*********************************************************************************************************)
FUNCTION_BLOCK FB_ASI_Projecting
VAR_INPUT
	iSlaveaddress		:BYTE;
	iParametervalue		:DWORD;
	bIOValue			:BOOL;	(*Read/Write IO-value of a slave*)
	bIDCode				:BOOL;	(*Read/Write	ID-code of a slave*)
	bReadWrite			:BOOL;	(*0: Read, 1: Write*)
	bReadLPS			:BOOL;	(*Read List of all projected Slaves*)
	bStart				:BOOL;
END_VAR
VAR_OUTPUT
	bBusy				:BOOL;
	bErr					:BOOL;
	iErrornumber			:DWORD;
	iParameterReadvalue	:BYTE;	(*IO-value or ID-code of a slave*)
	iLPS				:DWORD;
END_VAR
VAR_IN_OUT
	stParameterBuffer		:ST_ParameterBuffer;
END_VAR
VAR
	iProjectingStep	:INT;
	TrigStart			:R_TRIG;
	iAddressFactor	:BYTE;
	iParameternumber	:WORD;
	iReadValue		:DWORD;
	fbParameterinterface	:FB_ASI_Parameterinterface;
END_VAR
	CASE iProjectingStep OF

	(*Idle*)
	0:	TrigStart(clk:=bStart);
		IF TrigStart.Q THEN
			bBusy				:=TRUE;
			bErr					:=FALSE;
			iErrornumber			:=0;
			iProjectingStep		:=1;
		END_IF

	(*generate Parameternumber*)
	1:	iAddressFactor	:=iSlaveaddress / 8;
		IF bIOValue THEN
			iParameternumber	:=16#40+iAddressFactor;
		ELSIF bIDCode THEN
			iParameternumber	:=16#48+iAddressFactor;
		ELSIF bReadLPS	THEN
			iParameternumber	:=16#A8;
		END_IF
		iProjectingStep	:=2;

	(*write Parameter to ASI-Master*)
	2:	fbParameterinterface(iParameternumber	:=iParameternumber,
							iParametervalue	:=iParametervalue,
							stParameterBuffer	:=stParameterBuffer,
							bParametermode	:=bReadWrite,
							bCycleMode		:=TRUE,
							bStart			:=TRUE);
			IF (NOT fbParameterinterface.bBusy)  THEN
				IF fbParameterinterface.bErr THEN
					bErr			:=TRUE;
					iErrornumber	:=fbParameterinterface.iErrornumber;
					iProjectingStep	:=10;
				ELSE
					iReadValue	:=fbParameterinterface.iParameterReadvalue;
					iProjectingStep	:=3;
				END_IF
				fbParameterinterface(bStart			:=FALSE,
								stParameterBuffer	:=stParameterBuffer);
			END_IF

	(*generate ParameterReadvalue*)
	3:	IF bReadLPS THEN
			iParameterReadvalue	:=0;
			iLPS				:=iReadValue;
		ELSE
			iParameterReadvalue	:=DWORD_TO_BYTE(SHR(iReadValue,((iSlaveaddress-iAddressFactor*8)*4))) AND 2#00001111;
			iLPS	:=0;
		END_IF
		iProjectingStep	:=10;

	(*Quit*)
	10:	bBusy			:=FALSE;
		bStart			:=FALSE;
		iProjectingStep	:=0;

	ELSE
		;
	END_CASE
END_FUNCTION_BLOCK

(* POU FB_ASI_ReadParameter, ST *)
(*********************************************************************************************************

NAME..............	:	FB_ReadParameter
DATE...............	:	21.03.2002
AUTHOR........	:	G.Sieder (Beckhoff Industrieelektronik)

DESCRIPTION:	FB to read Parameters 

HISTORY:	
21.03.2002	gs	start coding

*********************************************************************************************************)
FUNCTION_BLOCK FB_ASI_ReadParameter
VAR_INPUT
	iParameternumber		:WORD;
	bCycleMode			:BOOL;		(*0: Acyclic , 1:Cyclic (permanent Read/Write) *)
	bStart				:BOOL;
END_VAR
VAR_OUTPUT
	bBusy				:BOOL;
	bErr					:BOOL;
	iErrornumber			:DWORD;
	iParameterReadvalue	:DWORD;
END_VAR
VAR_IN_OUT
	stParameterBuffer		:ST_ParameterBuffer;
END_VAR
VAR
	iReadStep	:INT;
	TrigStart		:R_TRIG;
	fbParameterinterface	:FB_ASI_Parameterinterface;
END_VAR
CASE iReadStep OF

	(*Idle*)
	0:	TrigStart(clk:=bStart);
		IF TrigStart.Q THEN
			bBusy				:=TRUE;
			bErr					:=FALSE;
			iErrornumber			:=0;
			iReadStep			:=1;
		END_IF

	(*wite Parameters to ASI-Master*)
	1:	fbParameterinterface(iParameternumber	:=iParameternumber,
							stParameterBuffer	:=stParameterBuffer,
							bParametermode	:=FALSE,
							bCycleMode		:=bCycleMode,
							bStart			:=TRUE);
		(*read Parameters *)
		IF (NOT fbParameterinterface.bBusy) OR  bCycleMode THEN
			IF fbParameterinterface.bErr THEN
				bErr			:=TRUE;
				iErrornumber	:=fbParameterinterface.iErrornumber;
				iReadStep	:=5;
			ELSE
				iParameterReadvalue	:=fbParameterinterface.iParameterReadvalue;
				IF (NOT bCycleMode) OR (NOT bStart) THEN
					iReadStep	:=5;
				ELSE
					iReadStep	:=1;
				END_IF
			END_IF
		END_IF

	5:	fbParameterinterface(bStart			:=FALSE,
						stParameterBuffer	:=stParameterBuffer);
		IF (NOT fbParameterinterface.bBusy) THEN
			iReadStep	:=10;
		END_IF

	(*Quit*)
	10:	bBusy			:=FALSE;
		bStart			:=FALSE;
		iReadStep	:=0;

	ELSE
		;
	END_CASE
END_FUNCTION_BLOCK

(* POU FB_ASI_SlaveDiag, ST *)
(*********************************************************************************************************

NAME..............	:	FB_WriteParameter
DATE...............	:	21.03.2002
AUTHOR........	:	G.Sieder (Beckhoff Industrieelektronik)

DESCRIPTION:	FB for cyclic slave-diagnosis

HISTORY:	
21.03.2002	gs	start coding
03.09.2002	gs	replace bStop by bCycleMode
*********************************************************************************************************)
FUNCTION_BLOCK FB_ASI_SlaveDiag
VAR_INPUT
	iSlaveaddress		:BYTE;
	iCounter				:INT;		(*1:PhysicalFaultCounter,  2:TimeoutCounter,  3:ResponseCounter,  4:Leave-DataExchCounter,  5:DataExch-FailedCounter *)
	bCounterReset		:BOOL;
	bReadLES			:BOOL;		(*Read List of all detected Slaves*)
	bReadLAS			:BOOL;		(*Read List of all activated Slaves*)
	bCycleMode			:BOOL;		(*0: Acyclic , 1:Cyclic (permanent Read/Write) *)
	bStart				:BOOL;

END_VAR
VAR_OUTPUT
	bBusy				:BOOL;
	bErr					:BOOL;
	iErrornumber			:DWORD;
	iCounterValue		:WORD;		(*Counter of a slave*)
	iSlaveList			:DWORD;	(*LES or LAS of all Slaves*)
END_VAR
VAR_IN_OUT
	stParameterBuffer		:ST_ParameterBuffer;
END_VAR
VAR
	iDiagStep			:INT;
	TrigStart				:R_TRIG;
	iAddressFactor		:BYTE;
	iParameternumber		:WORD;
	iReadValue			:DWORD;
	fbParameterinterface	:FB_ASI_Parameterinterface;

	TimerResetCounter	:TON;
END_VAR
	CASE iDiagStep OF

	(*Idle*)
	0:	TrigStart(clk:=bStart);
		IF TrigStart.Q THEN
			bBusy				:=TRUE;
			bErr					:=FALSE;
			iErrornumber			:=0;
			iDiagStep			:=1;
		END_IF

	(*generate Parameternumber*)
	1:	iAddressFactor	:=iSlaveaddress / 2;
		IF bReadLES	THEN
			iParameternumber	:=16#B0;
		ELSIF bReadLAS THEN
			iParameternumber	:=16#B8;
		ELSE
			CASE iCounter OF
				1:	iParameternumber	:=16#140+iAddressFactor;
				2:	iParameternumber	:=16#160+iAddressFactor;
				3:	iParameternumber	:=16#180+iAddressFactor;
				4:	iParameternumber	:=16#1A0+iAddressFactor;
				5:	iParameternumber	:=16#1C0+iAddressFactor;
			ELSE
				;
			END_CASE
		END_IF
		iDiagStep	:=2;

	(*write Parameter to ASI-Master*)
	2:	fbParameterinterface(iParameternumber		:=iParameternumber,
							stParameterBuffer		:=stParameterBuffer,
							iParametervalue		:=0,
							bParametermode		:=bCounterReset,
							bCycleMode			:=TRUE,
							bStart				:=TRUE);
				IF fbParameterinterface.bErr THEN
					bErr			:=TRUE;
					iErrornumber	:=fbParameterinterface.iErrornumber;
					iDiagStep	:=10;
				ELSE
					iReadValue	:=fbParameterinterface.iParameterReadvalue;
					iDiagStep	:=3;
				END_IF
				TimerResetCounter(in:=bCounterReset,pt:=t#200ms);
				IF TimerResetCounter.Q THEN
					bCounterReset		:=FALSE;
					TimerResetCounter.IN 	:=FALSE;
				END_IF

	(*generate ParameterReadvalue*)
	3:	fbParameterinterface(stParameterBuffer	:=stParameterBuffer);
		IF bReadLES OR bReadLAS THEN
			iCounterValue	:=0;
			iSlaveList		:=iReadValue;
		ELSE
			iCounterValue	:=DWORD_TO_WORD(SHR(iReadValue,((iSlaveaddress-iAddressFactor*2)*16)));
			iSlaveList	:=0;
		END_IF
		IF (NOT bStart) THEN
			fbParameterinterface(bStart	:=FALSE,
							stParameterBuffer	:=stParameterBuffer);
			IF (NOT fbParameterinterface.bBusy) THEN
				iDiagStep	:=10;
			END_IF
		ELSE
			iDiagStep	:=2;
		END_IF

	(*Quit*)
	10:	bBusy		:=FALSE;
		bStart		:=FALSE;
		iDiagStep	:=0;

	ELSE
		;
	END_CASE
END_FUNCTION_BLOCK

(* POU FB_ASI_WriteParameter, ST *)
(*********************************************************************************************************

NAME..............	:	FB_WriteParameter
DATE...............	:	21.03.2002
AUTHOR........	:	G.Sieder (Beckhoff Industrieelektronik)

DESCRIPTION:	FB to write Parameters 

HISTORY:	
21.03.2002	gs	start coding
03.09.2002	gs	Output ReadValue removed
*********************************************************************************************************)
FUNCTION_BLOCK FB_ASI_WriteParameter
VAR_INPUT
	iParameternumber		:WORD;
	iParametervalue		:DWORD;
	bStart				:BOOL;
END_VAR
VAR_OUTPUT
	bBusy				:BOOL;
	bErr					:BOOL;
	iErrornumber			:DWORD;
END_VAR
VAR_IN_OUT
	stParameterBuffer		:ST_ParameterBuffer;
END_VAR
VAR
	iWriteStep	:INT;
	TrigStart		:R_TRIG;
	fbParameterinterface	:FB_ASI_Parameterinterface;
END_VAR
	CASE iWriteStep OF

	(*Idle*)
	0:	TrigStart(clk:=bStart);
		IF TrigStart.Q THEN
			bBusy				:=TRUE;
			bErr					:=FALSE;
			iErrornumber			:=0;
			iWriteStep			:=1;
		END_IF

	(*wite Parameters to ASI-Master*)
	1:	fbParameterinterface(iParameternumber	:=iParameternumber,
							iParametervalue	:=iParametervalue,
							stParameterBuffer	:=stParameterBuffer,
							bParametermode	:=TRUE,
							bCycleMode		:= FALSE,
							bStart			:=TRUE);
		IF  fbParameterinterface.bBusy  THEN
			iWriteStep	:=5;
		END_IF


	5:	fbParameterinterface(stParameterBuffer	:=stParameterBuffer);
		IF (NOT fbParameterinterface.bBusy) THEN
			IF fbParameterinterface.bErr THEN
				bErr			:=TRUE;
				iErrornumber	:=fbParameterinterface.iErrornumber;
			END_IF
			iWriteStep	:=10;
		END_IF

	(*Quit*)
	10:	bBusy			:=FALSE;
		bStart			:=FALSE;
		iWriteStep	:=0;

	ELSE
		;
	END_CASE
END_FUNCTION_BLOCK

(* POU FB_ASI_WriteReadParameter, ST *)
(*********************************************************************************************************

NAME..............	:	FB_WriteReadParameter
DATE...............	:	18.08.2003
AUTHOR........	:	G.Sieder (Beckhoff Industrieelektronik)

DESCRIPTION:	FB to write Parameters with answer 

HISTORY:	
18.08.2003	gs	start coding

*********************************************************************************************************)
FUNCTION_BLOCK FB_ASI_WriteReadParameter
VAR_INPUT
	iParameternumber		:WORD;
	iParametervalue		:DWORD;
	bStart				:BOOL;
END_VAR
VAR_OUTPUT
	bBusy				:BOOL;
	bErr					:BOOL;
	iParameterReadValue	:DWORD;
	iErrornumber			:DWORD;
END_VAR
VAR_IN_OUT
	stParameterBuffer		:ST_ParameterBuffer;
END_VAR
VAR
	iWriteStep	:INT;
	TrigStart		:R_TRIG;
	fbParameterinterface	:FB_ASI_Parameterinterface;
END_VAR
	CASE iWriteStep OF

	(*Idle*)
	0:	TrigStart(clk:=bStart);
		IF TrigStart.Q THEN
			bBusy				:=TRUE;
			bErr					:=FALSE;
			iErrornumber			:=0;
			iWriteStep			:=1;
		END_IF

	(*wite Parameters to ASI-Master*)
	1:	fbParameterinterface(iParameternumber	:=iParameternumber,
							iParametervalue	:=iParametervalue,
							stParameterBuffer	:=stParameterBuffer,
							bParametermode	:=TRUE,
							bCycleMode		:= FALSE,
							bStart			:=TRUE);
		IF  fbParameterinterface.bBusy  THEN
			iWriteStep	:=5;
		END_IF


	5:	fbParameterinterface(stParameterBuffer	:=stParameterBuffer);
		IF (NOT fbParameterinterface.bBusy) THEN
			IF fbParameterinterface.bErr THEN
				bErr			:=TRUE;
				iErrornumber	:=fbParameterinterface.iErrornumber;
				iParameterReadValue	:=0;
			ELSE
				iParameterReadValue	:=fbParameterinterface.iParameterReadvalue;
			END_IF
			iWriteStep	:=10;
		END_IF

	(*Quit*)
	10:	bBusy			:=FALSE;
		bStart			:=FALSE;
		iWriteStep	:=0;

	ELSE
		;
	END_CASE
END_FUNCTION_BLOCK

(* POU FB_AX2000_AXACT, ST *)
FUNCTION_BLOCK FB_AX2000_AXACT
VAR_INPUT
	bMode_DigitalSpeed	: BOOL;			(*OP-Mode digital speed instead of Positioning*)
	iDigitalSpeed			: DWORD;			(*digital speed if OP-Mode = digital speed*)
	iVelocity				: DWORD;		(*Velocity*)
	iPosition				: DINT;			(*Position*)
	imotion_tasknumber	: WORD;			(*number of EEPROM-saved motion-task*)
	imotion_blocktype		: WORD;			(*optional Parameters of motion tasks*)
	bStart				: BOOL;			(*START*)
	bStop				: BOOL;			(*STOP*)
	bShortStop			: BOOL;			(*1: break of motion task, 0: continue same motion task*)
	bErrorResume		: BOOL;			(*Error resume*)
	tTimeOut				: TIME:=t#5s;
END_VAR
VAR_OUTPUT

	bBusy				: BOOL;
	bError				: BOOL;			(*Errorstatus of Servo*)
	bTimeOutErr			: BOOL;

END_VAR
VAR
	i16State:				INT;
	icheckStatus:			WORD;
	icheckControlWord:	WORD;			(*ControlWord for Servo*)

	bServoReady:		BOOL;			(*readyFlag for HSW*)
	TrigStart:				R_TRIG;
	TrigTimeOut:			R_TRIG;
	bResetServo:			BOOL;			(*first move of Servo after Start/Restart*)

	TimerTimeOut		:TON;
	bTimeOutStart		:BOOL;

	iHighByte			:BYTE;
	iLowByte				:BYTE;
	icheckByteSwaping	:WORD;
	bMapInOutputs		:BOOL;
	bShortStop_check		:BOOL;

	(*virtual Input/Output*)
	stPZD_IN:		ST_PZD_IN;
	stPZD_OUT:		ST_PZD_OUT;
END_VAR
VAR_IN_OUT
	stPZDIN:		ST_PZD_IN;			(*Data from NC*)
	stPZDOUT:		ST_PZD_OUT;			(*Data to NC*)
END_VAR
	a_MapInputs();			(*mapping of real Inputs to virtual Inputs by swaping LowByte and HighByte*)
	a_RW_CtrlWord();			(*AXACT-controls*)
	a_MapOutputs();			(*mapping of virtual Outputs to real Outputs by swaping LowByte and HighByte*)
END_FUNCTION_BLOCK
ACTION a_MapInputs:
stPZD_IN.wSTW		:=ROL(stPZDIN.wSTW,8);
stPZD_IN.wHIW		:=ROL(stPZDIN.wHIW,8);
stPZD_IN.PZD3		:=ROL(stPZDIN.PZD3,8);
stPZD_IN.PZD4		:=ROL(stPZDIN.PZD4,8);
stPZD_IN.PZD5		:=ROL(stPZDIN.PZD5,8);
stPZD_IN.PZD6		:=ROL(stPZDIN.PZD6,8);
END_ACTION
ACTION a_MapOutputs:
IF bMapInOutputs THEN
	stPZDOUT.wCtrlW		:=ROL(stPZD_OUT.wCtrlW,8);
	stPZDOUT.PZD2		:=ROL(stPZD_OUT.PZD2,8);
	stPZDOUT.PZD3		:=ROL(stPZD_OUT.PZD3,8);
	stPZDOUT.PZD4		:=ROL(stPZD_OUT.PZD4,8);
	stPZDOUT.PZD5		:=ROL(stPZD_OUT.PZD5,8);
	stPZDOUT.PZD6		:=ROL(stPZD_OUT.PZD6,8);
END_IF
END_ACTION
ACTION a_RW_CtrlWord:
	bMapInOutputs	:= TRUE;

	(* Errorstatus*)
	icheckStatus:=2#00000000_00001000;
	IF (stPZD_IN.wSTW AND icheckStatus)<>0 THEN
		i16State:=10;
	END_IF

	(*short break of a motion task*)
	IF bShortStop AND (NOT bShortStop_check)THEN
		stPZD_OUT.wCtrlW:=stPZD_OUT.wCtrlW AND 2#1111111111011111;
		bShortStop_check	:=TRUE;
	ELSIF (NOT bShortStop) AND bShortStop_check THEN
		bShortStop_check	:=FALSE;
		IF (NOT bStart) THEN
			i16State			:= 11;
			bBusy			:= FALSE;
		ELSE
			stPZD_OUT.wCtrlW:=stPZD_OUT.wCtrlW OR 2#0000000000100000;
		END_IF
	END_IF

	(*Stophandling*)
	IF  bStop THEN
		stPZD_OUT.wCtrlW:=2#0000000000000101;
		bBusy			:= FALSE;
		bStart			:= FALSE;
		bMapInOutputs	:= TRUE;
		i16State			:= 11;
	END_IF

	(*TimeOut*)
	IF (NOT bMode_DigitalSpeed) THEN
		TrigTimeOut(clk:=bStart);
		IF TrigTimeOut.Q THEN
			bTimeOutStart	:=TRUE;
			bTimeOutErr		:= FALSE;
			bError			:= FALSE;
		END_IF
		IF bBusy THEN
			TimerTimeOut(IN:= FALSE, PT:= tTimeOut );
			bTimeOutStart	:=FALSE;
		ELSE
			TimerTimeOut(IN:= bTimeOutStart, PT:= tTimeOut );
		END_IF
		IF TimerTimeOut.Q THEN
			bTimeOutErr		:=TRUE;
			bTimeOutStart	:= FALSE;
			bServoReady	:= FALSE;
			i16State			:= 11;
		END_IF
	END_IF

	CASE i16State OF

		(*Initialisierung*)
	0:	bServoReady:= 	FALSE;
		bResetServo:=	TRUE;
		i16State:= i16State+1;

		(*Einschaltsperre*)
	1:	stPZD_OUT.wCtrlW:=2#0000000000000000;
		icheckStatus:=2#0000000001000000;
		IF (stPZD_IN.wSTW AND icheckStatus)<>0 THEN
			stPZD_OUT.wCtrlW:=2#0000000000000110;
			bServoReady:= FALSE;
			i16State:= i16State+1;
		END_IF

		(*einschaltbereit*)
	2:	icheckStatus:=2#0000001000000001;
		IF (stPZD_IN.wSTW AND icheckStatus)<>0 THEN
			stPZD_OUT.wCtrlW:=2#0000000000000111;
			bServoReady:= FALSE;
			i16State:= i16State+1;
		END_IF

		(*betriebsbereit*)
	3:	icheckStatus:=2#0000001000100011;
		IF (stPZD_IN.wSTW AND icheckStatus)<>0 THEN
			stPZD_OUT.wCtrlW:=2#0000010000111111;
			i16State:= i16State+1;
		END_IF

		(*Betrieb freigegeben*)
	4:	icheckStatus:=2#0000001000100111;
		IF (stPZD_IN.wSTW AND icheckStatus)<>0 THEN
			i16State:= i16State+1;
		END_IF

		(*benutzerdefinierte Daten übertragen*)
	5:	TrigStart(clk:=bStart);
		bMapInOutputs	:= FALSE;
		IF TrigStart.Q THEN
			bMapInOutputs:= TRUE;
			a_RW_PZD();
			bError		:= FALSE;
			bTimeOutErr	:= FALSE;
			bResetServo	:= FALSE;
		END_IF
		IF (NOT bResetServo) THEN
			icheckStatus:=2#0010000000000000;
			IF (stPZD_IN.wSTW AND icheckStatus)<>0 THEN
				;
			ELSE
				bBusy	:= TRUE;
				i16State:= 6;
			END_IF
		END_IF

	6:	icheckStatus:=2#0010000000000000;
		IF (stPZD_IN.wSTW AND icheckStatus)<>0 THEN
			bBusy	:= FALSE;
			i16State:= 5;
		END_IF
		IF bMode_DigitalSpeed THEN
			stPZD_OUT.PZD3	:=DWORD_TO_WORD(iDigitalSpeed*140);
			stPZD_OUT.PZD2	:=DWORD_TO_WORD(SHR((iDigitalSpeed*140),16));
		END_IF

		(* Errorhandling*)
	10:	bError			:= TRUE;
		bBusy			:= FALSE;
		bServoReady	:= FALSE;
		IF BErrorResume THEN
			stPZD_OUT.wCtrlW:=2#0000010010001111;
			i16State:=11;
		END_IF

	11:	IF (NOT bStart) THEN
			i16State:=0;
		END_IF

END_CASE
END_ACTION
ACTION a_RW_PZD:
IF bMode_DigitalSpeed THEN
	stPZD_OUT.PZD3	:=DWORD_TO_WORD(iDigitalSpeed*140);
	stPZD_OUT.PZD2	:=DWORD_TO_WORD(SHR((iDigitalSpeed*140),16));
	icheckControlWord:=2#0000000001000000;
	IF (icheckControlWord AND stPZD_OUT.wCtrlW)<>0 THEN
		stPZD_OUT.wCtrlW:=16#443F;
	ELSE
		stPZD_OUT.wCtrlW:=16#447F;
	END_IF
ELSIF (imotion_tasknumber <> 0) THEN
	stPZD_OUT.PZD2	:=imotion_tasknumber;
	icheckControlWord:=2#0000000001000000;
	IF (icheckControlWord AND stPZD_OUT.wCtrlW)<>0 THEN
		stPZD_OUT.wCtrlW:=16#043F;
	ELSE
		stPZD_OUT.wCtrlW:=16#047F;
	END_IF
ELSIF (iVelocity<>0) THEN
	stPZD_OUT.PZD3	:=DWORD_TO_WORD(iVelocity);
	stPZD_OUT.PZD2	:=DWORD_TO_WORD(SHR(iVelocity,16));
	stPZD_OUT.PZD5	:=DWORD_TO_WORD(DINT_TO_DWORD( iPosition ));
	stPZD_OUT.PZD4	:=DWORD_TO_WORD(SHR(DINT_TO_DWORD( iPosition ),16));
	stPZD_OUT.PZD6	:=imotion_blocktype;
	icheckControlWord:=2#0000000001000000;
	IF (icheckControlWord AND stPZD_OUT.wCtrlW)<>0 THEN
		stPZD_OUT.wCtrlW:=16#443F;
	ELSE
		stPZD_OUT.wCtrlW:=16#447F;
	END_IF
END_IF
END_ACTION

(* POU FB_AX2000_JogMode, ST *)
FUNCTION_BLOCK FB_AX2000_JogMode
VAR_INPUT
	bStart		: BOOL;
	bStop		: BOOL;
	iBasicVelo	: INT;				(*BasicVelocity*)
	tTimeOut		: TIME:=t#5s;

END_VAR
VAR_OUTPUT
	bBusy		: BOOL;
	bErr			: BOOL;
	bTimeOutErr	: BOOL;

END_VAR
VAR_IN_OUT
	stPZDIN			: ST_PZD_IN;			(*Data from NC*)
	stPZDOUT		: ST_PZD_OUT;		(*Data to NC*)
END_VAR
VAR
	i16state			: INT;

	icheckStatus		: DWORD;
	TrigTimeOut		: R_TRIG;
	bTimeOutStart	: BOOL;
	TimerTimeOut	: TON;
	bMapInOutputs	: BOOL;
	(*virtual Input/Output*)
	stPZD_IN:		ST_PZD_IN;
	stPZD_OUT:		ST_PZD_OUT;

END_VAR
	a_MapInputs();

	(* Errorstatus*)
	icheckStatus:=2#00000000_00001000;
	IF (stPZD_IN.wSTW AND icheckStatus)<>0 THEN
		bErr	:= TRUE;
		i16State:=10;
	END_IF

	(*TimeOut*)
	TrigTimeOut(clk:=bStart);
	IF TrigTimeOut.Q THEN
		bTimeOutStart	:=TRUE;
	END_IF
	IF bBusy THEN
		TimerTimeOut(IN:= FALSE, PT:= tTimeOut );
		bTimeOutStart	:=FALSE;
	ELSE
		TimerTimeOut(IN:= bTimeOutStart, PT:= tTimeOut );
	END_IF
	IF TimerTimeOut.Q THEN
		TimerTimeOut(IN:= FALSE, PT:= tTimeOut );
		bTimeOutErr		:=TRUE;
		bTimeOutStart	:= FALSE;
		i16State			:= 10;
	END_IF

	CASE i16state OF

	0:	IF bStart THEN
			bErr				:= FALSE;
			bTimeOutErr		:= FALSE;
			i16state			:= 1;
		END_IF

	1:	stPZD_OUT.PZD2	:=iBasicVelo;
		stPZD_OUT.wCtrlW:=(ROL(stPZDOUT.wCtrlW,8))+16#100;
		bMapInOutputs	:= TRUE;
		i16state	:= 2;

	2:	icheckStatus:=2#00100010_00000000;
		IF (stPZD_IN.wSTW AND icheckStatus)=0 OR  (stPZD_IN.wSTW AND icheckStatus)=16#2200 THEN
			;
		ELSE
			bBusy	:=TRUE;
			i16state	:= 3;
		END_IF

	3:	IF bStop THEN
			stPZD_OUT.wCtrlW:=(ROL(stPZDOUT.wCtrlW,8))-16#100;
			i16state	:= 10;
		END_IF

	10:	bBusy			:=FALSE;
		bMapInOutputs	:=FALSE;
		IF (NOT bstart) THEN
			i16state	:= 0;
		END_IF

	END_CASE

	a_MapOutputs();
END_FUNCTION_BLOCK
ACTION a_MapInputs:
	stPZD_IN.wSTW		:=ROL(stPZDIN.wSTW,8);
	stPZD_IN.wHIW		:=ROL(stPZDIN.wHIW,8);
	stPZD_IN.PZD3		:=ROL(stPZDIN.PZD3,8);
	stPZD_IN.PZD4		:=ROL(stPZDIN.PZD4,8);
	stPZD_IN.PZD5		:=ROL(stPZDIN.PZD5,8);
	stPZD_IN.PZD6		:=ROL(stPZDIN.PZD6,8);
END_ACTION
ACTION a_MapOutputs:
IF bMapInOutputs THEN
	stPZDOUT.wCtrlW		:=ROL(stPZD_OUT.wCtrlW,8);
	stPZDOUT.PZD2		:=ROL(stPZD_OUT.PZD2,8);
	stPZDOUT.PZD3		:=ROL(stPZD_OUT.PZD3,8);
	stPZDOUT.PZD4		:=ROL(stPZD_OUT.PZD4,8);
	stPZDOUT.PZD5		:=ROL(stPZD_OUT.PZD5,8);
	stPZDOUT.PZD6		:=ROL(stPZD_OUT.PZD6,8);
END_IF
END_ACTION

(* POU FB_AX2000_Parameter, ST *)
FUNCTION_BLOCK FB_AX2000_Parameter
VAR_INPUT
	iSlaveAddress:	BYTE := 0;			(* Station Address of the Slave *)
	iPnu:				WORD := 16#03A2;	(* Parameter-Number *)
	nAxis:				BYTE := 1;			(* Number of Axis *)
	iLength:			BYTE := 4;			(* Length of the parameter (2 or 4) *)
	iSubindex:			BYTE := 1;			(*Subindex*)
	iParameterValue:	DWORD := 2;			(* Parameter value *)
	iFC310xDeviceId: 	WORD := 1;			(* Device-ID of the FCxxxx *)
	bStartRead:		BOOL;				(* StartFlag to start the PKW-Read *)
	bStartWrite:		BOOL;				(* StartFlag to start the PKW-Write *)
	tTimeOut:			TIME := DEFAULT_ADS_TIMEOUT;
END_VAR
VAR_OUTPUT
	bBusy				:BOOL;
	iErrorId			:DWORD;
	iReadValue		:DINT;
END_VAR
VAR
	iError:					DWORD;
	fbReadPkw:				FB_FCxxxxDpv0PkwRead;
	fbWritePkw: 				FB_FCxxxxDpv0PkwWrite;

END_VAR
IF bStartRead OR bStartWrite THEN
	IF iLength<>2 THEN
		iLength:= 4;
	END_IF
	
	(* PKW-Read with DPV0  for Stoever-Drive (ArrayCodesNotSupported and Subindex in Octet 3 must be set) *)
	fbReadPkw(bStartFlag := bStartRead, iStationAdd := iSlaveAddress, iDeviceId := iFC310xDeviceId,nAxis := nAxis, iPnu := iPnu, iSubindex := iSubindex, iLength := iLength, bArrayCodesNotSupported := TRUE, bSubindexInOctet3 := TRUE, tTimeOut:=tTimeOut);
	IF (bStartRead AND NOT fbReadPkw.bBusy) THEN
		iError := fbReadPkw.iErrorId;
		iReadValue := fbReadPkw.iReadValue;
		bStartRead := FALSE;
	END_IF;
	
	(* PKW-Write with DPV0  for Stoever-Drive (ArrayCodesNotSupported and Subindex in Octet 3 must be set) *)
	fbWritePkw(bStartFlag := bStartWrite, iStationAdd := iSlaveAddress, iDeviceId := iFC310xDeviceId, nAxis := nAxis, iPnu := iPnu, iSubindex := iSubindex, iLength := iLength, iWriteValue := iParameterValue, bArrayCodesNotSupported := TRUE, bSubindexInOctet3 := TRUE, tTimeOut:=tTimeOut);
	IF (bStartWrite AND NOT fbWritePkw.bBusy) THEN
		iError := fbWritePkw.iErrorId;
		bStartWrite := FALSE;
	END_IF;

	bBusy:=fbReadPkw.bBusy OR fbWritePkw.bBusy;
	iErrorId:=iError;
	(*iReadValue:=iParameterValue;*)
END_IF
END_FUNCTION_BLOCK

(* POU FB_FCxxxxDpv0PkwRead, ST *)
FUNCTION_BLOCK FB_FCxxxxDpv0PkwRead
VAR_INPUT
	bStartFlag:BOOL;					(* StartFlag to start the PKW-Read *)
	iStationAdd: BYTE;				(* Station Address of the Slave *)
	iDeviceId: WORD;					(* Device-ID of the FCxxxx *)
	nAxis: BYTE;						(* Number of Axis *)
	iPnu: WORD;						(* Parameter-Number *)
	iSubindex: BYTE;					(* Subindex  *)
	iLength:BYTE;					(* Length of the parameter (2 or 4) *)
	bArrayCodesNotSupported: BOOL;	(* if the drive does not support the ARRAY-AKs 6,7 and 8, this flag should be set (then the AKs 1,2,3 will be used for Arrays) *)
	bSubindexInOctet3:BOOL;			(* if the drive needs the subindex in Octet 3 (ProfiDrive 2.0), this flag should be set *)
	tTimeOut		: TIME;
END_VAR
VAR_OUTPUT
	bBusy:BOOL;			(* Reading is busy *)
	iErrorId:DWORD;
	iReadValue:DWORD;	(* Parameter value *)
END_VAR
VAR
	fbRead:ADSREAD;
	fbDevNetId:IOF_GetDeviceNetId;
	istate:WORD := 0;
	sDevNetId:STRING(23);
	iIdxGrp: DWORD;
	iport:WORD;
	iParameterValue:DWORD;
END_VAR
CASE istate OF

	0:	(*Idle*)
		IF bStartFlag THEN
			bBusy	:=TRUE;
			istate := 1;
		END_IF

	1:	(* Get Net-ID of FCxxxx-Device *)
		fbDevNetId(NETID := '', DEVICEID := iDeviceId, START := TRUE,  TMOUT := T#1s);
		IF (NOT fbDevNetId.BUSY) THEN
			IF (NOT fbDevNetId.Err) THEN
				sDevNetId := fbDevNetId.DeviceNetId;
				istate := 2;
			ELSE
				iErrorId		:=fbDevNetId.ERRID;
				bStartFlag	:=FALSE;
				bBusy		:=FALSE;
				istate := 0;
			END_IF
			fbDevNetId(NETID := '', DEVICEID := iDeviceId, START := FALSE,  TMOUT := T#1s);
		END_IF

	2:	(* Read Parameter if StartFlag is set *)
		iport := iStationAdd;
		iport := iport + 16#1000;
		iIdxGrp := nAxis;
		iIdxGrp := SHL(iIdxGrp, 28);
		iIdxGrp := iIdxGrp +iPnu;
		IF (bArrayCodesNotSupported) THEN
			iIdxGrp := iIdxGrp + 16#8000000;
		END_IF
		IF (bSubindexInOctet3) THEN
			iIdxGrp := iIdxGrp + 16#4000000;
		END_IF
		fbRead(	NETID := sDevNetId, PORT := iport, IDXGRP := iIdxGrp, IDXOFFS := iSubindex, LEN := iLength,
				DESTADDR := ADR(iParameterValue), READ := bStartFlag, TMOUT := tTimeOut);
		istate := 3;

	3:	fbRead(	NETID := sDevNetId, PORT := iport, IDXGRP := iIdxGrp, IDXOFFS := iSubindex, LEN := iLength,
				DESTADDR := ADR(iParameterValue), READ := bStartFlag, TMOUT := tTimeOut);
		IF (NOT FbRead.BUSY) OR fbRead.Err THEN
			iErrorId := FbRead.ERRID;
			iReadValue := iParameterValue;
			istate := 4;
		END_IF

	4:	(* There must be a rising edge on the READ-input of ADSREAD to start the next reading *)
		fbRead(	NETID := sDevNetId, PORT := iport, IDXGRP := iIdxGrp, IDXOFFS := iSubindex, LEN := iLength,
				DESTADDR := ADR(iParameterValue), READ := FALSE, TMOUT := tTimeOut);
		bBusy 		:= FALSE;
		bStartFlag	:= FALSE;
		istate := 0;
END_CASE
END_FUNCTION_BLOCK

(* POU IOF_GetDeviceNetId, ST *)
FUNCTION_BLOCK IOF_GetDeviceNetId
VAR_INPUT
	NETID			: T_AmsNetId;
	DEVICEID		: UDINT;
	START			: BOOL;
	TMOUT		: TIME := DEFAULT_ADS_TIMEOUT;
END_VAR
VAR_OUTPUT
	BUSY			: BOOL;
	ERR			: BOOL;
	ERRID			: UDINT;
	DeviceNetId	: T_AmsNetId;
END_VAR
VAR
	ADSREADEX1	: ADSREADEX;
	RisingEdge	: R_TRIG;
	state			: BYTE;
	tmpNetId		: ARRAY[0..5] OF BYTE;
END_VAR
RisingEdge( CLK:=START );
IF RisingEdge.Q THEN
	state := 1;
END_IF
CASE state OF
	0:;(* idle state *)
	1:
		BUSY := TRUE;
		ERR := FALSE;
		ERRID := 0;
		DeviceNetId := '';
		MEMSET( ADR( tmpNetId ), 0, SIZEOF( tmpNetId ) );
		IF ( DEVICEID > 0 ) THEN
			ADSREADEX1( READ:=FALSE );
			ADSREADEX1( NETID:=NETID, PORT:= AMSPORT_R0_IO,
						IDXGRP:= 16#00005000 + DEVICEID, IDXOFFS:= 16#00000005,
						LEN:= SIZEOF( tmpNetId ), DESTADDR:= ADR( tmpNetId ),
						READ:=TRUE, TMOUT:= TMOUT );
			state := 2;
		ELSE
			ERR := TRUE;
			ERRID :=16#706;	(* Parameter value not correct! *)
			state := 100;
		END_IF
	2:
		ADSREADEX1( READ:=FALSE, BUSY=>BUSY, ERR=>ERR, ERRID=>ERRID );
		IF NOT BUSY THEN
			IF NOT ERR THEN
				IF ( ADSREADEX1.COUNT_R = SIZEOF( tmpNetId ) ) THEN (* check the read data length *)
					DeviceNetId := F_CreateAmsNetId( tmpNetid );
				ELSE
					ERR := TRUE;
					ERRID := 16#70B; (* 1803 invalid parameter value(s) *)
				END_IF
			END_IF
			state := 0;
		END_IF
	100:(* error state *)
		BUSY := FALSE;
		state := 0;
END_CASE
END_FUNCTION_BLOCK

(* POU FB_FCxxxxDpv0PkwWrite, ST *)
FUNCTION_BLOCK FB_FCxxxxDpv0PkwWrite
VAR_INPUT
	bStartFlag:BOOL;		(* StartFlag to start the PKW-REad *)
	iStationAdd: BYTE;		(* Station Address of the Slave *)
	iDeviceId: WORD;		(* Device-ID of the FCxxxx *)
	nAxis: BYTE;			(* Number of Axis *)
	iPnu: WORD;			(* Parameter-Number *)
	iSubindex: BYTE;		(* Subindex  *)
	iLength:BYTE;			(* Length of the parameter (2 or 4) *)
	iWriteValue:DWORD;	(* Parameter value *)
	bArrayCodesNotSupported: BOOL;	(* if the drive does not support the ARRAY-AKs 6,7 and 8, this flag should be set (then the AKs 1,2,3 will be used for Arrays) *)
	bSubindexInOctet3:BOOL;				(* if the drive needs the subindex in Octet 3 (ProfiDrive 2.0), this flag should be set *)
	tTimeOut		: TIME:=T#10s;
END_VAR
VAR_OUTPUT
	bBusy:BOOL;			(* Writing is busy *)
	iErrorId:DWORD;
END_VAR
VAR
	fbWrite:ADSWRITE;
	fbDevNetId:IOF_GetDeviceNetId;
	istate:WORD := 0;
	sDevNetId:STRING(23);
	iIdxGrp: DWORD;
	iport:WORD;
	iParameterValue:DWORD;
END_VAR
CASE istate OF

	0:	(*Idle*)
		IF bStartFlag THEN
			bBusy	:=TRUE;
			istate := 1;
		END_IF

	1:	(* Get Net-ID of FCxxxx-Device *)
		fbDevNetId(NETID := '', DEVICEID :=iDeviceId, START := TRUE,  TMOUT := T#1s);
		istate := 2;

	2:	fbDevNetId();
		IF (NOT fbDevNetId.BUSY) THEN
			IF (NOT fbDevNetId.Err) THEN
				sDevNetId := fbDevNetId.DeviceNetId;
				istate := 3;
			ELSE
				iErrorId		:=fbDevNetId.ERRID;
				bBusy		:=FALSE;
				bStartFlag	:=FALSE;
				istate := 0;
			END_IF
			fbDevNetId(NETID := '', DEVICEID := iDeviceId, START := FALSE,  TMOUT := T#1s);
		END_IF

	3:	(* Read Parameter if StartFlag is set *)
		iport := iStationAdd;
		iport := iport + 16#1000;
		iIdxGrp :=nAxis;
		iIdxGrp := SHL(iIdxGrp, 28);
		iIdxGrp := iIdxGrp + iPnu;
		IF (bArrayCodesNotSupported) THEN
			iIdxGrp := iIdxGrp + 16#8000000;
		END_IF
		IF (bSubindexInOctet3) THEN
			iIdxGrp := iIdxGrp + 16#4000000;
		END_IF
		iParameterValue :=iWriteValue;
		fbWrite(	NETID := sDevNetId, PORT := iport, IDXGRP := iIdxGrp, IDXOFFS := iSubindex, LEN := iLength,
				SRCADDR := ADR(iParameterValue), WRITE := bStartFlag, TMOUT := tTimeOut);
		istate := 4;

	4:	fbWrite();
		IF (NOT fbWrite.BUSY) OR fbWrite.Err THEN
			iErrorId := fbWrite.ERRID;
			istate := 5;
		END_IF

	5:	(* There must be a rising edge on the READ-input of ADSREAD to start the next reading *)
		fbWrite(	NETID := sDevNetId, PORT := iport, IDXGRP := iIdxGrp, IDXOFFS := iSubindex, LEN := iLength,
				SRCADDR := ADR(iParameterValue), WRITE := FALSE, TMOUT := tTimeOut);
		bBusy 		:= FALSE;
		bStartFlag	:= FALSE;
		istate := 0;
END_CASE
END_FUNCTION_BLOCK

(* POU FB_AX2000_Reference, ST *)
FUNCTION_BLOCK FB_AX2000_Reference
VAR_INPUT
	bSetRefPoint	: BOOL;		(* set Reference Point*)
	bCalibrStart	: BOOL;		(* start home running*)
	bCalibrStop	: BOOL;		(* stop home running*)
	iCalVelo		: WORD;		(* basic velocity of Calibration*)

END_VAR
VAR_OUTPUT
	bBusy	: BOOL;
	bErr	: BOOL;

END_VAR
VAR_IN_OUT
	stPZDIN		: ST_PZD_IN;	(*Data from NC*)
	stPZDOUT		: ST_PZD_OUT;(*Data to NC*)
END_VAR
VAR
	icheckStatus		: WORD;
	i16State			: INT;
	bMapInOutputs	: BOOL;
	(*virtual Input/Output*)
	stPZD_IN		: ST_PZD_IN;	(*Data from NC*)
	stPZD_OUT		: ST_PZD_OUT;(*Data to NC*)
END_VAR
	a_MapInputs();

	(* Errorstatus*)
	icheckStatus:=2#00000000_00001000;
	IF (stPZD_IN.wSTW AND icheckStatus)<>0 THEN
		i16State	:=9;
	END_IF

	CASE i16State OF

	(*start FB*)
	0:	IF bSetRefPoint OR bCalibrStart THEN
			bBusy			:= TRUE;
			bErr				:= FALSE;
			IF bSetRefPoint THEN
				i16State	:= 1;
			ELSE
				i16State	:= 3;
			END_IF
		END_IF

	(* set Reference Point *)
	1:	bMapInOutputs	:=TRUE;
		(*realization of a rising edge to set a nwe reference point*)
		stPZD_OUT.wCtrlW:=(ROL(stPZDOUT.wCtrlW,8))-16#1000;
		i16State		:= 2;

	2:	stPZD_OUT.wCtrlW:=(ROL(stPZDOUT.wCtrlW,8))+16#1000;
		i16State		:= 10;

	(* start home running*)
	3:	bMapInOutputs	:=TRUE;
		stPZD_OUT.PZD2	:=iCalVelo;
		(*stPZD_OUT.wCtrlW:=(ROL(stPZDOUT.wCtrlW,8))+16#800;*)
		stPZD_OUT.wCtrlW:=((ROL(stPZDOUT.wCtrlW,8)) OR 2#0000100000000000);
		icheckStatus:=2#0000010000000000;
		IF (stPZD_IN.wSTW AND icheckStatus)<>0 THEN
			(*Stophandling*)
			IF bCalibrStop THEN
				(*stPZD_OUT.wCtrlW:=(ROL(stPZDOUT.wCtrlW,8))-16#800;*)
				stPZD_OUT.wCtrlW:=((ROL(stPZDOUT.wCtrlW,8)) AND 2#1111011111111111);
				i16State	:= 10;
			ELSE
				;
			END_IF
		ELSE
			i16State:=4;
		END_IF

	4:	icheckStatus:=2#0000010000000000;
		IF ((stPZD_IN.wSTW AND icheckStatus)<>0)  THEN
			i16State	:= 10;
		END_IF
		(*Stophandling*)
		IF bCalibrStop THEN
			stPZD_OUT.wCtrlW:=(ROL(stPZDOUT.wCtrlW,8))-16#800;
			i16State	:= 10;
		END_IF

		(*Errorcase*)
	9:	bErr			:= TRUE;
		i16State		:= 10;

	10:	bbusy			:= FALSE;
		bMapInOutputs	:= FALSE;
		bSetRefPoint		:= FALSE;
		IF (NOT bSetRefPoint) AND (NOT bCalibrStart) THEN
			i16State	:= 0;
		END_IF

	END_CASE

	a_MapOutputs();
END_FUNCTION_BLOCK
ACTION a_MapInputs:
	stPZD_IN.wSTW		:=ROL(stPZDIN.wSTW,8);
	stPZD_IN.wHIW		:=ROL(stPZDIN.wHIW,8);
	stPZD_IN.PZD3		:=ROL(stPZDIN.PZD3,8);
	stPZD_IN.PZD4		:=ROL(stPZDIN.PZD4,8);
	stPZD_IN.PZD5		:=ROL(stPZDIN.PZD5,8);
	stPZD_IN.PZD6		:=ROL(stPZDIN.PZD6,8);
END_ACTION
ACTION a_MapOutputs:
IF bMapInOutputs THEN
	stPZDOUT.wCtrlW		:=ROL(stPZD_OUT.wCtrlW,8);
	stPZDOUT.PZD2		:=ROL(stPZD_OUT.PZD2,8);
	stPZDOUT.PZD3		:=ROL(stPZD_OUT.PZD3,8);
	stPZDOUT.PZD4		:=ROL(stPZD_OUT.PZD4,8);
	stPZDOUT.PZD5		:=ROL(stPZD_OUT.PZD5,8);
	stPZDOUT.PZD6		:=ROL(stPZD_OUT.PZD6,8);
END_IF
END_ACTION

(* POU FB_AX200X_Profibus, ST *)
FUNCTION_BLOCK FB_AX200X_Profibus
VAR_INPUT
	bInit					: BOOL;			(*Initialization*)
	bMode_DigitalSpeed	: BOOL;			(*OP-Mode digital speed instead of Positioning*)
	iDigitalSpeed			: DINT;			(*digital speed if OP-Mode = digital speed*)
	iVelocity				: DWORD;		(*Velocity*)
	iPosition				: DINT;			(*Position*)
	iRunningMode		: BYTE;			(*0:digital speed, 1: motiontask, 2: JogMode, 3: Calibration*)
	imotion_tasknumber	: WORD;			(*number of EEPROM-saved motion-task*)
	imotion_blocktype		: WORD:=16#2000;	(*optional Parameters of motion tasks, default:SI-values*)
	iJogModeBasicValue	: INT;			(*BasicVelocity for JogMode*)
	iCalVelo				: WORD;			(* basic velocity of Calibration*)
	bSetRefPoint			: BOOL;			(* set Reference Point*)
	bStart					: BOOL;			(*START*)
	bStop					: BOOL;			(*STOP*)
	bShortStop			: BOOL;			(* break of motion task*)
	iSlaveAddress			: BYTE;			(* Station Address of the Slave *)
	iFC310xDeviceId 		: WORD;			(* Device-ID of the FCxxxx *)
	bErrorResume		: BOOL;			(*Error resume*)
	tTimeOut				: TIME := DEFAULT_ADS_TIMEOUT;
END_VAR
VAR_OUTPUT

	bBusy				: BOOL;
	bError				: BOOL;			(*Errorstatus of Servo*)
	iErrID				: DWORD;
	bTimeOutErr		: BOOL;
	bInitOK			: BOOL;				(*Initialization OK*)
	iactPosition		 : DINT;		(*actual Position SI-value*)
END_VAR
VAR_IN_OUT
	stPZD_IN:			ST_PZD_IN;				(*Data from NC*)
	stPZD_OUT:			ST_PZD_OUT;			(*Data to NC*)
END_VAR
VAR
	istate					:INT;
	TimerPosition				:TON;
	fbAX2000_AXACT			: FB_AX2000_AXACT;
	fbAX2000_Parameter		: FB_AX2000_Parameter;
	fbAX2000_JogMode		: FB_AX2000_JogMode;
	fbAX2000_Reference		: FB_AX2000_Reference;

	iOPMode				:DWORD;
END_VAR
VAR CONSTANT
	(*Errors*)
	ERR_OPMODE	:DWORD:=1;

END_VAR
		fbAX2000_AXACT(bMode_DigitalSpeed	:=bMode_DigitalSpeed,
						iDigitalSpeed			:=iDigitalSpeed,
						iVelocity				:=iVelocity,
						 iPosition				:=iPosition ,
						 imotion_tasknumber	:=imotion_tasknumber ,
						 imotion_blocktype	:=imotion_blocktype ,
						bShortStop			:=bShortStop,
						 bErrorResume		:=bErrorResume ,
						 tTimeOut			:=tTimeOut ,
						stPZDIN				:= stPZD_IN,
						stPZDOUT			:=stPZD_OUT);
	IF iRunningMode<2 OR bInit THEN
			fbAX2000_AXACT.bStart	:=bStart;
	END_IF

	IF (NOT bInit) THEN
		fbAX2000_AXACT.bStop	:=bStop;
	END_IF

	IF fbAX2000_AXACT.stPZD_IN.wSTW =0 THEN
		bInitOK	:=FALSE;
	END_IF

	CASE istate OF

	(*action-mode*)
	0:	(*Initialization*)
		IF bInit THEN
			bBusy		:=TRUE;
			bError		:=FALSE;
			bTimeOutErr	:=FALSE;
			iErrID		:=0;
			bInitOK		:=FALSE;
			IF bMode_DigitalSpeed THEN
				iOPMode	:= 1;
			ELSE
				iOPMode	:= 2;
			END_IF
			istate		:=1;
		(*JogMode*)
		ELSIF iRunningMode=2 AND bStart THEN
			IF bInitOK THEN
				bBusy		:=TRUE;
				bError		:=FALSE;
				bTimeOutErr	:=FALSE;
				iErrID		:=0;
				istate		:=20;
			ELSE
				iErrID	:=ERR_OPMODE;
				istate	:=100;
			END_IF
		(*CalibrationMode*)
		ELSIF iRunningMode=3 AND (bStart OR  bSetRefPoint)THEN
			IF bInitOK THEN
				bBusy		:=TRUE;
				bError		:=FALSE;
				bTimeOutErr	:=FALSE;
				iErrID		:=0;
				istate		:=30;
			ELSE
				iErrID	:=ERR_OPMODE;
				istate	:=100;
			END_IF
		(*motion-task start*)
		ELSIF (iRunningMode=1 OR iRunningMode=0) AND bStart  THEN
			IF bInitOK THEN
				bBusy		:=TRUE;
				bError		:=FALSE;
				bTimeOutErr	:=FALSE;
				iErrID		:=0;
				istate		:=10;
			ELSE
				iErrID	:=ERR_OPMODE;
				istate	:=100;
			END_IF
		ELSIF iRunningMode>3 AND bStart  THEN
			iErrID	:=ERR_OPMODE;
			istate	:=100;
		END_IF

	(*Init*)
	1:	fbAX2000_AXACT.bStop	:=TRUE;
		istate	:=2;

	2:	fbAX2000_Parameter(iSlaveAddress:= iSlaveAddress,
						iPnu:= 930,
						iParameterValue:= iOPMode,
						iFC310xDeviceId:=iFC310xDeviceId ,
						bStartWrite:= TRUE );
		istate	:=3;

	3:	fbAX2000_Parameter();
		IF (NOT fbAX2000_Parameter.bBusy) THEN
			IF fbAX2000_Parameter.iErrorId<>0 THEN
				iErrID	:=fbAX2000_Parameter.iErrorId;
				bInit		:=FALSE;
				istate	:=100;
			ELSE
				istate	:=4;
			END_IF
			fbAX2000_AXACT.bStop	:=FALSE;
		END_IF

	4:	fbAX2000_Parameter(iSlaveAddress:= iSlaveAddress,
						iPnu:= 930,
						iFC310xDeviceId:=iFC310xDeviceId ,
						bStartRead:= TRUE );
		istate	:=5;

	5:	fbAX2000_Parameter();
		IF (NOT fbAX2000_Parameter.bBusy)  THEN
			IF fbAX2000_Parameter.iErrorId<>0 THEN
				iErrID	:=fbAX2000_Parameter.iErrorId;
				istate	:=100;
			ELSE
				bInitOK	:=TRUE;
				istate	:=110;
			END_IF
			bInit		:=FALSE;
		END_IF

	(*motion task start*)
	10:	IF fbAX2000_AXACT.bBusy THEN
			istate	:=11;
		ELSIF fbAX2000_AXACT.bError THEN
			fbAX2000_Parameter(iSlaveAddress:= iSlaveAddress,
							iPnu:= 1001,
							iFC310xDeviceId:=iFC310xDeviceId ,
							bStartRead:= TRUE );
			iErrID	:=fbAX2000_Parameter.iReadValue;
			istate	:=100;
		ELSIF fbAX2000_AXACT.bTimeOutErr  THEN
			bTimeOutErr	:=TRUE;
			istate	:=100;
		END_IF

	11:	fbAX2000_Parameter(iSlaveAddress:= iSlaveAddress,
						iPnu:= 1403,
						iFC310xDeviceId:=iFC310xDeviceId ,
						bStartRead:= TRUE);
		iactPosition	:=fbAX2000_Parameter.iReadValue;
		IF (NOT fbAX2000_AXACT.bBusy) THEN
			TimerPosition(in:=TRUE, PT:=t#1s);
			IF TimerPosition.Q THEN
				TimerPosition(in:=FALSE);
				istate	:=12;
			END_IF
		END_IF

	12:	fbAX2000_Parameter();
		iactPosition	:=fbAX2000_Parameter.iReadValue;
		IF (NOT fbAX2000_Parameter.bBusy) THEN
			istate	:=110;
		END_IF

	(*JogMode*)
	20:	fbAX2000_JogMode(bStart:= bStart,
						bStop		:= bStop,
						 iBasicVelo	:=iJogModeBasicValue,
						 tTimeOut	:=tTimeOut ,
						stPZDIN		:= stPZD_IN,
						stPZDOUT	:=stPZD_OUT);
		fbAX2000_Parameter(iSlaveAddress:= iSlaveAddress,
						iPnu:= 1403,
						iFC310xDeviceId:=iFC310xDeviceId ,
						bStartRead:= TRUE);
		iactPosition	:=fbAX2000_Parameter.iReadValue;
		IF bStop OR fbAX2000_JogMode.bErr OR fbAX2000_JogMode.bTimeOutErr THEN
			istate	:=21;
		END_IF

	21:	fbAX2000_Parameter();
		iactPosition	:=fbAX2000_Parameter.iReadValue;
		IF (NOT fbAX2000_Parameter.bBusy) THEN
			bStart		:= FALSE;
			fbAX2000_JogMode(bStart		:= bStart,
							bStop		:= FALSE,
							 iBasicVelo	:=iJogModeBasicValue,
							 tTimeOut	:=tTimeOut ,
							stPZDIN		:= stPZD_IN,
							stPZDOUT	:=stPZD_OUT);
			istate	:=110;
			IF fbAX2000_JogMode.bErr THEN
				fbAX2000_Parameter(iSlaveAddress:= iSlaveAddress,
								iPnu:= 1001,
								iFC310xDeviceId:=iFC310xDeviceId ,
								bStartRead:= TRUE );
				iErrID	:=fbAX2000_Parameter.iReadValue;
				istate	:=100;
			ELSIF fbAX2000_JogMode.bTimeOutErr THEN
				bTimeOutErr	:=TRUE;
			END_IF
		END_IF

	(*CalibrationMode*)
	30:	fbAX2000_Reference(bSetRefPoint	:= bSetRefPoint ,
						bCalibrStart		:= bStart,
						bCalibrStop		:= bStop,
						iCalVelo			:= iCalVelo,
						stPZDIN			:= stPZD_IN,
						stPZDOUT		:=stPZD_OUT);
		fbAX2000_Parameter(iSlaveAddress:= iSlaveAddress,
						iPnu:= 1403,
						iFC310xDeviceId:=iFC310xDeviceId ,
						bStartRead:= TRUE);
		iactPosition	:=fbAX2000_Parameter.iReadValue;
		IF bStop OR fbAX2000_Reference.bErr  THEN
			istate	:=31;
		END_IF

	31:	fbAX2000_Parameter();
		iactPosition	:=fbAX2000_Parameter.iReadValue;
		IF (NOT fbAX2000_Parameter.bBusy) THEN
			bStart		:= FALSE;
			fbAX2000_Reference(bCalibrStart	:= bStart,
							bCalibrStop		:= TRUE,
							stPZDIN			:= stPZD_IN,
							stPZDOUT		:=stPZD_OUT);
			istate	:=110;
			IF fbAX2000_Reference.bErr THEN
				fbAX2000_Parameter(iSlaveAddress:= iSlaveAddress,
								iPnu:= 1001,
								iFC310xDeviceId:=iFC310xDeviceId ,
								bStartRead:= TRUE );
				iErrID	:=fbAX2000_Parameter.iReadValue;
				istate	:=100;
			END_IF
		END_IF


	(*Error*)
	100:	bError	:=TRUE;
		istate	:=110;

	(*Quit*)
	110:	bBusy	:=FALSE;
		IF (NOT bStart) AND (NOT bInit) THEN
			istate	:=0;
		END_IF


	ELSE
		;
	END_CASE
END_FUNCTION_BLOCK

(* POU FB_Dpv1Read, ST *)
FUNCTION_BLOCK FB_Dpv1Read
(*****************************************************************************************************************
	DESCRIPTION:	This FUNCTION block implements DPV1 Parameter Read

	CHANGE LOG:
	BY		DATE		DESCRIPTION OF CHANGE
	ICh		2008/04/02	delay resend request after fault for 100ms
	ICh		2007/01/08	resend request after fault
	ICh		2007/01/05	iRequestRef limited to 128
	ICh		2006/08/09	wait timer decreased, bugfix for errors
	ICh		2006/07/12	Bugfix iRequestRef as VAR_IN_OUT
	ICh		2006/07/10	Bugfix for evaluate response; enhanced error reporting
	ICh		2006/07/05	First Version

******************************************************************************************************************)
VAR_INPUT
	bExecute			: BOOL;

	(* drive access info *)
	aNetId				: T_AmsNetId;	(* NetID of Profibus Master FC310x/EL6731 *)
	iProfibusSlaveAdr	: USINT;	 	(* DP address of ProfiDrive *)
	iDriveId			: USINT;		(* 0..255 possible *)
	pDpv1ReqData		: POINTER TO ARRAY [1..iMAX_DPV1_SIZE] OF BYTE;
	iDpv1ReqDataLen		: UDINT;
	pDpv1ResData		: POINTER TO ARRAY [1..iMAX_DPV1_SIZE] OF BYTE;
	iDpv1ResDataLen		: UDINT;
	tTmOut				: TIME := DEFAULT_ADS_TIMEOUT;
END_VAR
VAR_OUTPUT
	bBusy				: BOOL;
	bError				: BOOL;
	bErrorValues		: BOOL;
	iErrId				: UDINT;
	iErrorClass			: BYTE;
	iErrorCode			: BYTE;
END_VAR
VAR_IN_OUT
	iRequestRef			: USINT;		(* 1..127;    0: reserved *)
END_VAR
VAR
	fbWriteAccessData 	: ADSWRITE;
	fbReadData 			: ADSREAD;
	iState				: INT;
	bExecute_			: BOOL;

	stDpv1ReqHeader		: ST_Dpv1Header;
	stDpv1ResHeader		: ST_Dpv1Header;

	WaitTimer			: TON := (PT := T#100ms);
	TmOutTimer			: TON;
END_VAR
TmOutTimer();

CASE iState OF
0:	(* idle until rising edge on bExecute *)
	IF bExecute AND NOT bExecute_ THEN
		(* generate request reference *)
		iRequestRef := UINT_TO_USINT((USINT_TO_UINT(iRequestRef) + 1) MOD 128);
		IF iRequestRef = 0 THEN
			iRequestRef := 1;
		END_IF
		pDpv1ReqData^[1] := iRequestRef;
		MEMCPY(ADR(stDpv1ReqHeader), pDpv1ReqData, SIZEOF(stDpv1ReqHeader));

		(* clear response data *)
		MEMSET(pDpv1ResData, 0, iMAX_DPV1_SIZE);

		(* on rising edge *)
		bExecute_ 	:= bExecute;
		bBusy		:= TRUE;
		bError		:= FALSE;
		bErrorValues:= FALSE;
		iErrId		:= 0;
		iErrorClass	:= 0;
		iErrorCode	:= 0;

		(* complete read request timeout 12 times the ADS timeout *)
		TmOutTimer(IN := FALSE, PT := MAX(tTmOut * 12, T#30s));
		TmOutTimer(IN := TRUE);

		(* send request *)
		fbWriteAccessData(
			NETID	:= aNetId,
			PORT	:= 16#1000 + iProfibusSlaveAdr,
			IDXGRP	:= 0,
			IDXOFFS	:= 47,
			LEN		:= MIN(iDpv1ReqDataLen, iMAX_DPV1_SIZE),
			SRCADDR	:= pDpv1ReqData,
			WRITE	:= FALSE,
			TMOUT	:= tTmOut
		);
		fbWriteAccessData(WRITE	:= TRUE);

		iState := 1;
	END_IF

1:	(* write access data for DPV1 read request *)
	fbWriteAccessData(WRITE	:= FALSE);

	IF NOT fbWriteAccessData.BUSY THEN
		fbWriteAccessData(WRITE	:= FALSE);

		IF NOT fbWriteAccessData.ERR THEN
			(* read request parameter successfully sent, check for response *)
			WaitTimer(IN := FALSE);
			iState	:= 2; (* wait before polling *)
		ELSE
			bBusy	:= FALSE;
			bError	:= TRUE;
			iErrId	:= fbWriteAccessData.ERRID;
			IF ((UDINT_TO_DWORD(iErrId) AND DWORD#16#FF000000) = DWORD#16#27000000) THEN
				iErrorClass := UDINT_TO_BYTE(SHR((UDINT_TO_DWORD(iErrId) AND 16#00F00000), 20));
				iErrorCode := UDINT_TO_BYTE(SHR((UDINT_TO_DWORD(iErrId) AND 16#000F0000), 16));
			END_IF
			iState	:= 0;
		END_IF
	END_IF

2:	(* wait staate before next read response check *)
	WaitTimer(IN := TRUE);
	IF WaitTimer.Q THEN
		(* read request parameter successfully sent, check for read response *)
		MEMSET(pDpv1ResData, 0, iMAX_DPV1_SIZE);
		fbReadData(
			NETID	:= aNetId,
			PORT	:= 16#1000 + iProfibusSlaveAdr,
			IDXGRP	:= 0,
			IDXOFFS	:= 47,
			LEN		:= iMAX_DPV1_SIZE,
			DESTADDR:= pDpv1ResData,
			READ	:= FALSE,
			TMOUT	:= tTmOut,
		);
		fbReadData(READ := TRUE);
		iState	:= 3; (* CHECK READ *)
	END_IF

3:	(* wait for read response with data from DPV1 read request *)
	fbReadData(READ := FALSE);

	IF NOT fbReadData.BUSY THEN
		fbReadData(READ := FALSE);
		IF NOT fbReadData.ERR THEN
			MEMCPY(ADR(stDpv1ResHeader), pDpv1ResData, SIZEOF(stDpv1ResHeader));

			(* check for read response reference *)
			IF (stDpv1ResHeader.iRequestRef = stDpv1ReqHeader.iRequestRef) AND (stDpv1ResHeader.iAxis = stDpv1ReqHeader.iAxis) THEN
				(* response to last parameter request - split response data *)
				TmOutTimer(IN := FALSE);
				iState	:= 5;	(* DONE *)
			ELSIF stDpv1ResHeader.iRequestRef = 0 THEN
				(* no response *)
				IF TmOutTimer.Q THEN
					(* complete read request timed out *)
					TmOutTimer(IN := FALSE);
					bBusy	:= FALSE;
					bError	:= TRUE;
					iErrId	:= 16#745; (* timeout *)
					iState	:= 0; (* ERROR *)
				ELSE
					(* no response, go to wait state *)
					WaitTimer(IN := FALSE);
					iState	:= 2; (* WAIT and REPEAT *)
				END_IF
			ELSE
				(* wrong response *)
				bBusy	:= FALSE;
				bError	:= TRUE;
				iErrId	:= 2; (* wrong reference response *)
				iState	:= 0; (* ERROR *)
			END_IF
		ELSE
			IF ((UDINT_TO_DWORD(fbReadData.ERRID) AND DWORD#16#FFFF0000) = DWORD#16#27B50000) THEN
				(* repeat telegram *)
				WaitTimer(IN := FALSE);
				iState	:= 4; (* SEND NEW REQUEST *)
			ELSE
				(* error *)
				bBusy	:= FALSE;
				bError	:= TRUE;
				iErrId	:= fbReadData.ERRID;
				IF ((UDINT_TO_DWORD(iErrId) AND DWORD#16#FF000000) = DWORD#16#27000000) THEN
					iErrorClass := UDINT_TO_BYTE(SHR((UDINT_TO_DWORD(iErrId) AND 16#00F00000), 20));
					iErrorCode := UDINT_TO_BYTE(SHR((UDINT_TO_DWORD(iErrId) AND 16#000F0000), 16));
				END_IF
				iState	:= 0; (* ERROR *)
			END_IF
		END_IF
	END_IF

4:	(* generate new request reference after fault *)
	WaitTimer(IN := TRUE);
	IF WaitTimer.Q THEN
		iRequestRef := UINT_TO_USINT((USINT_TO_UINT(iRequestRef) + 1) MOD 128);
		IF iRequestRef = 0 THEN
			iRequestRef := 1;
		END_IF
		pDpv1ReqData^[1] := iRequestRef;
		MEMCPY(ADR(stDpv1ReqHeader), pDpv1ReqData, SIZEOF(stDpv1ReqHeader));
	
		(* clear response data *)
		MEMSET(pDpv1ResData, 0, iMAX_DPV1_SIZE);
	
		(* send request *)
		fbWriteAccessData(
			NETID	:= aNetId,
			PORT	:= 16#1000 + iProfibusSlaveAdr,
			IDXGRP	:= 0,
			IDXOFFS	:= 47,
			LEN		:= MIN(iDpv1ReqDataLen, iMAX_DPV1_SIZE),
			SRCADDR	:= pDpv1ReqData,
			WRITE	:= FALSE,
			TMOUT	:= tTmOut
		);
		fbWriteAccessData(WRITE	:= TRUE);
	
		iState := 1; (* CHECK WRITE *)
	END_IF

5:	(* evaluate response *)
	IF stDpv1ResHeader.iRequestID = stDpv1ReqHeader.iRequestID THEN
		(* DPV1 Read successful - done *)
		bBusy	:= FALSE;
		iState	:= 0; (* DONE *)
	ELSIF (SINT_TO_BYTE(stDpv1ResHeader.iRequestID) AND 16#7F) = SINT_TO_BYTE(stDpv1ReqHeader.iRequestID) THEN
		(* DPV1 Read not successful or partly not successful *)
		bErrorValues:= TRUE;
		bBusy	:= FALSE;
		bError	:= TRUE;
		iErrId	:= 3; (* DPV1 Read not successful or partly not successful *)
		iState	:= 0; (* ERROR *)
	ELSE
		(* wrong response *)
		bBusy	:= FALSE;
		bError	:= TRUE;
		iErrId	:= 4; (* wrong response ID *)
		iState	:= 0; (* ERROR *)
	END_IF

END_CASE

(* clear flag *)
bExecute_ := bExecute_ AND bExecute;
END_FUNCTION_BLOCK

(* POU FB_Dpv1ReadPNET, ST *)
FUNCTION_BLOCK FB_Dpv1ReadPNET
(*****************************************************************************************************************
	DESCRIPTION:	This FUNCTION block implements DPV1 Parameter Read for Profinet

	CHANGE LOG:
	BY		DATE		DESCRIPTION OF CHANGE
	ICh		2009/07/23	First Version

******************************************************************************************************************)
VAR_INPUT
	bExecute			: BOOL;

	(* drive access info *)
	aNetId				: T_AmsNetId;	(* NetID of Profibus Master EL6631 *)
	iProfinetPort		: UINT;		 	(* Port of ProfiDrive *)
	iDriveId			: USINT;		(* 0..255 possible *)
	pDpv1ReqData		: POINTER TO ARRAY [1..iMAX_DPV1_SIZE_PNET_REQ] OF BYTE;
	iDpv1ReqDataLen		: UDINT;
	pDpv1ResData		: POINTER TO ARRAY [1..iMAX_DPV1_SIZE_PNET_RES] OF BYTE;
	iDpv1ResDataLen		: UDINT;
	tTmOut				: TIME;
END_VAR
VAR_OUTPUT
	bBusy				: BOOL;
	bError				: BOOL;
	bErrorValues		: BOOL;
	iErrId				: UDINT;
	iErrorClass			: BYTE;
	iErrorCode			: BYTE;
END_VAR
VAR_IN_OUT
	iRequestRef			: USINT;		(* 1..127;    0: reserved *)
END_VAR
VAR
	fbRWData 			: ADSRDWRT;
	iState				: INT;
	bExecute_			: BOOL;
	iIGrp				: UDINT := 16#F823;
	stDpv1ReqHeader		: ST_Dpv1Header;
	stDpv1ResHeader		: ST_Dpv1Header;
	stPNETFrameHeader	: ST_PNIOConfigRecord;

	WaitTimer			: TON := (PT := T#100ms);
	TmOutTimer			: TON;
END_VAR
TmOutTimer();

CASE iState OF
0:	(* idle until rising edge on bExecute *)
	IF bExecute AND NOT bExecute_ THEN
		(* generate request reference *)
		iRequestRef := UINT_TO_USINT((USINT_TO_UINT(iRequestRef) + 1) MOD 128);
		IF iRequestRef = 0 THEN
			iRequestRef := 1;
		END_IF
		pDpv1ReqData^[1] := 1; pDpv1ReqData^[2] := 0; (* write request *)
		pDpv1ReqData^[1+SIZEOF(stPNETFrameHeader)] := iRequestRef;
		MEMCPY(ADR(stPNETFrameHeader), pDpv1ReqData, SIZEOF(stPNETFrameHeader));
		MEMCPY(ADR(stDpv1ReqHeader), pDpv1ReqData+SIZEOF(stPNETFrameHeader), SIZEOF(stDpv1ReqHeader));

		(* clear response data *)
		MEMSET(pDpv1ResData, 0, iMAX_DPV1_SIZE_PNET_RES);

		(* on rising edge *)
		bExecute_ 	:= bExecute;
		bBusy		:= TRUE;
		bError		:= FALSE;
		bErrorValues:= FALSE;
		iErrId		:= 0;
		iErrorClass	:= 0;
		iErrorCode	:= 0;

		(* complete read request timeout 12 times the ADS timeout *)
		TmOutTimer(IN := FALSE, PT := MAX(tTmOut * 12, T#30s));
		TmOutTimer(IN := TRUE);

		(* send request *)
		fbRWData(
			NETID	:= aNetId,
			PORT	:= iProfinetPort,
			IDXGRP	:= iIGrp,
			IDXOFFS	:= 0,
			WRITELEN:= MIN(iDpv1ReqDataLen, iMAX_DPV1_SIZE_PNET_REQ),
			SRCADDR	:= pDpv1ReqData,
			READLEN	:= MIN(iDpv1ResDataLen, iMAX_DPV1_SIZE_PNET_RES),
			DESTADDR:= pDpv1ResData,
			WRTRD	:= FALSE,
			TMOUT	:= tTmOut
		);
		fbRWData(WRTRD	:= TRUE);
		iState := 1;
	END_IF

1:	(* write access data for DPV1 read request *)
	fbRWData(WRTRD	:= FALSE);

	IF NOT fbRWData.BUSY THEN
		fbRWData(WRTRD	:= FALSE);

		IF NOT fbRWData.ERR THEN
			(* read request parameter successfully sent, check for response *)
			WaitTimer(IN := FALSE);
			iState	:= 2; (* wait before polling *)
		ELSE
			bBusy	:= FALSE;
			bError	:= TRUE;
			iErrId	:= fbRWData.ERRID;
			IF ((UDINT_TO_DWORD(iErrId) AND DWORD#16#FF000000) = DWORD#16#27000000) THEN
				iErrorClass := UDINT_TO_BYTE(SHR((UDINT_TO_DWORD(iErrId) AND 16#00F00000), 20));
				iErrorCode := UDINT_TO_BYTE(SHR((UDINT_TO_DWORD(iErrId) AND 16#000F0000), 16));
			END_IF
			iState	:= 0;
		END_IF
	END_IF

2:	(* wait staate before next read response check *)
	WaitTimer(IN := TRUE);
	IF WaitTimer.Q THEN
		stPNETFrameHeader.iRW := 0; (* read response *)
		stPNETFrameHeader.stPNIORecord.iLength := UDINT_TO_INT(MIN(iDpv1ResDataLen, iMAX_DPV1_SIZE_PNET_RES)); (* max read response length *)

		(* read request parameter successfully sent, check for read response *)
		MEMSET(pDpv1ResData, 0, iMAX_DPV1_SIZE_PNET_RES);
		fbRWData(
			NETID	:= aNetId,
			PORT	:= iProfinetPort,
			IDXGRP	:= iIGrp,
			IDXOFFS	:= 0,
			WRITELEN:= SIZEOF(stPNETFrameHeader),
			SRCADDR	:= ADR(stPNETFrameHeader),
			READLEN	:= MIN(iDpv1ResDataLen, iMAX_DPV1_SIZE_PNET_RES),
			DESTADDR:= pDpv1ResData,
			WRTRD	:= FALSE,
			TMOUT	:= tTmOut
		);
		fbRWData(WRTRD	:= TRUE);
		iState	:= 3; (* CHECK READ *)
	END_IF

3:	(* wait for read response with data from DPV1 read request *)
	fbRWData(WRTRD	:= FALSE);

	IF NOT fbRWData.BUSY THEN
		fbRWData(WRTRD := FALSE);
		IF NOT fbRWData.ERR THEN
			MEMCPY(ADR(stDpv1ResHeader), pDpv1ResData, SIZEOF(stDpv1ResHeader));

			(* check for read response reference *)
			IF (stDpv1ResHeader.iRequestRef = stDpv1ReqHeader.iRequestRef) AND (stDpv1ResHeader.iAxis = stDpv1ReqHeader.iAxis) THEN
				(* response to last parameter request - split response data *)
				TmOutTimer(IN := FALSE);
				iState	:= 5;	(* DONE *)
			ELSIF stDpv1ResHeader.iRequestRef = 0 THEN
				(* no response *)
				IF TmOutTimer.Q THEN
					(* complete read request timed out *)
					TmOutTimer(IN := FALSE);
					bBusy	:= FALSE;
					bError	:= TRUE;
					iErrId	:= 16#745; (* timeout *)
					iState	:= 0; (* ERROR *)
				ELSE
					(* no response, go to wait state *)
					WaitTimer(IN := FALSE);
					iState	:= 2; (* WAIT and REPEAT *)
				END_IF
			ELSE
				(* wrong response *)
				bBusy	:= FALSE;
				bError	:= TRUE;
				iErrId	:= 2; (* wrong reference response *)
				iState	:= 0; (* ERROR *)
			END_IF
		ELSE
			IF ((UDINT_TO_DWORD(fbRWData.ERRID) AND DWORD#16#FFFF0000) = DWORD#16#27B50000) THEN
				(* repeat telegram *)
				WaitTimer(IN := FALSE);
				iState	:= 4; (* SEND NEW REQUEST *)
			ELSE
				(* error *)
				bBusy	:= FALSE;
				bError	:= TRUE;
				iErrId	:= fbRWData.ERRID;
				IF ((UDINT_TO_DWORD(iErrId) AND DWORD#16#FF000000) = DWORD#16#27000000) THEN
					iErrorClass := UDINT_TO_BYTE(SHR((UDINT_TO_DWORD(iErrId) AND 16#00F00000), 20));
					iErrorCode := UDINT_TO_BYTE(SHR((UDINT_TO_DWORD(iErrId) AND 16#000F0000), 16));
				END_IF
				iState	:= 0; (* ERROR *)
			END_IF
		END_IF
	END_IF

4:	(* generate new request reference after fault *)
	WaitTimer(IN := TRUE);
	IF WaitTimer.Q THEN
		iRequestRef := UINT_TO_USINT((USINT_TO_UINT(iRequestRef) + 1) MOD 128);
		IF iRequestRef = 0 THEN
			iRequestRef := 1;
		END_IF
		pDpv1ReqData^[1] := 1; pDpv1ReqData^[2] := 0; (* write request *)
		pDpv1ReqData^[1+SIZEOF(stPNETFrameHeader)] := iRequestRef;
		MEMCPY(ADR(stPNETFrameHeader), pDpv1ReqData, SIZEOF(stPNETFrameHeader));
		MEMCPY(ADR(stDpv1ReqHeader), pDpv1ReqData+SIZEOF(stPNETFrameHeader), SIZEOF(stDpv1ReqHeader));

		(* clear response data *)
		MEMSET(pDpv1ResData, 0, iMAX_DPV1_SIZE_PNET_RES);

		(* send request *)
		fbRWData(
			NETID	:= aNetId,
			PORT	:= iProfinetPort,
			IDXGRP	:= iIGrp,
			IDXOFFS	:= 0,
			WRITELEN:= MIN(iDpv1ReqDataLen, iMAX_DPV1_SIZE_PNET_REQ),
			SRCADDR	:= pDpv1ReqData,
			READLEN	:= MIN(iDpv1ResDataLen, iMAX_DPV1_SIZE_PNET_RES),
			DESTADDR:= pDpv1ResData,
			WRTRD	:= FALSE,
			TMOUT	:= tTmOut
		);
		fbRWData(WRTRD	:= TRUE);

		iState := 1; (* CHECK WRITE *)
	END_IF

5:	(* evaluate response *)
	IF stDpv1ResHeader.iRequestID = stDpv1ReqHeader.iRequestID THEN
		(* DPV1 Read successful - done *)
		bBusy	:= FALSE;
		iState	:= 0; (* DONE *)
	ELSIF (SINT_TO_BYTE(stDpv1ResHeader.iRequestID) AND 16#7F) = SINT_TO_BYTE(stDpv1ReqHeader.iRequestID) THEN
		(* DPV1 Read not successful or partly not successful *)
		bErrorValues:= TRUE;
		bBusy	:= FALSE;
		bError	:= TRUE;
		iErrId	:= 3; (* DPV1 Read not successful or partly not successful *)
		iState	:= 0; (* ERROR *)
	ELSE
		(* wrong response *)
		bBusy	:= FALSE;
		bError	:= TRUE;
		iErrId	:= 4; (* wrong response ID *)
		iState	:= 0; (* ERROR *)
	END_IF

END_CASE

(* clear flag *)
bExecute_ := bExecute_ AND bExecute;
END_FUNCTION_BLOCK

(* POU FB_Dpv1Write, ST *)
FUNCTION_BLOCK FB_Dpv1Write
(*****************************************************************************************************************
	DESCRIPTION:	This FUNCTION block implements DPV1 Parameter Write

	CHANGE LOG:
	BY		DATE		DESCRIPTION OF CHANGE
	ICh		2008/04/02	delay resend request after fault for 100ms
	ICh		2007/01/08	resend request after fault
	ICh		2007/01/05	iRequestRef limited to 128
	ICh		2006/08/09	wait timer decreased, bugfix for errors
	ICh		2006/07/12	Bugfix iRequestRef as VAR_IN_OUT
	ICh		2006/07/10	Bugfix for evaluate response; enhanced error reporting
	ICh		2006/07/07	First Version

******************************************************************************************************************)
VAR_INPUT
	bExecute			: BOOL;

	(* drive access info *)
	aNetId				: T_AmsNetId;	(* NetID of Profibus Master FC310x/EL6731 *)
	iProfibusSlaveAdr	: USINT;	 	(* DP address of ProfiDrive *)
	iDriveId			: USINT;		(* 0..255 possible *)
	pDpv1ReqData		: POINTER TO ARRAY [1..iMAX_DPV1_SIZE] OF BYTE;
	iDpv1ReqDataLen		: UDINT;
	pDpv1ResData		: POINTER TO ARRAY [1..iMAX_DPV1_SIZE] OF BYTE;
	iDpv1ResDataLen		: UDINT;
	tTmOut				: TIME := DEFAULT_ADS_TIMEOUT;
END_VAR
VAR_OUTPUT
	bBusy				: BOOL;
	bError				: BOOL;
	bErrorValues		: BOOL;
	iErrId				: UDINT;
	iErrorClass			: BYTE;
	iErrorCode			: BYTE;
END_VAR
VAR_IN_OUT
	iRequestRef			: USINT;		(* 1..127;    0: reserved *)
END_VAR
VAR
	fbWriteAccessData 	: ADSWRITE;
	fbReadData 			: ADSREAD;
	iState				: INT;
	bExecute_			: BOOL;

	stDpv1ReqHeader		: ST_Dpv1Header;
	stDpv1ResHeader		: ST_Dpv1Header;

	WaitTimer			: TON := (PT := T#100ms);
	TmOutTimer			: TON;
END_VAR
TmOutTimer();

CASE iState OF
0:	(* idle until rising edge on bExecute *)
	IF bExecute AND NOT bExecute_ THEN
		(* generate request reference *)
		iRequestRef := UINT_TO_USINT((USINT_TO_UINT(iRequestRef) + 1) MOD 128);
		IF iRequestRef = 0 THEN
			iRequestRef := 1;
		END_IF
		pDpv1ReqData^[1] := iRequestRef;
		MEMCPY(ADR(stDpv1ReqHeader), pDpv1ReqData, SIZEOF(stDpv1ReqHeader));

		(* clear response data *)
		MEMSET(pDpv1ResData, 0, iMAX_DPV1_SIZE);

		(* on rising edge *)
		bExecute_ 	:= bExecute;
		bBusy		:= TRUE;
		bError		:= FALSE;
		bErrorValues:= FALSE;
		iErrId		:= 0;
		iErrorClass	:= 0;
		iErrorCode	:= 0;

		(* complete read request timeout 12 times the ADS timeout *)
		TmOutTimer(IN := FALSE, PT := MAX(tTmOut * 12, T#30s));
		TmOutTimer(IN := TRUE);

		(* send request *)
		fbWriteAccessData(
			NETID	:= aNetId,
			PORT	:= 16#1000 + iProfibusSlaveAdr,
			IDXGRP	:= 0,
			IDXOFFS	:= 47,
			LEN		:= MIN(iDpv1ReqDataLen, iMAX_DPV1_SIZE),
			SRCADDR	:= pDpv1ReqData,
			WRITE	:= FALSE,
			TMOUT	:= tTmOut
		);
		fbWriteAccessData(WRITE	:= TRUE);

		iState := 1;
	END_IF

1:	(* write access data for DPV1 read request *)
	fbWriteAccessData(WRITE	:= FALSE);

	IF NOT fbWriteAccessData.BUSY THEN
		fbWriteAccessData(WRITE	:= FALSE);

		IF NOT fbWriteAccessData.ERR THEN
			(* read request parameter successfully sent, check for response *)
			WaitTimer(IN := FALSE);
			iState	:= 2; (* wait before polling *)
		ELSE
			bBusy	:= FALSE;
			bError	:= TRUE;
			iErrId	:= fbWriteAccessData.ERRID;
			IF ((UDINT_TO_DWORD(iErrId) AND DWORD#16#FF000000) = DWORD#16#27000000) THEN
				iErrorClass := UDINT_TO_BYTE(SHR((UDINT_TO_DWORD(iErrId) AND 16#00F00000), 20));
				iErrorCode := UDINT_TO_BYTE(SHR((UDINT_TO_DWORD(iErrId) AND 16#000F0000), 16));
			END_IF
			iState	:= 0;
		END_IF
	END_IF

2:	(* wait staate before next read response check *)
	WaitTimer(IN := TRUE);
	IF WaitTimer.Q THEN
		(* read request parameter successfully sent, check for read response *)
		MEMSET(pDpv1ResData, 0, iMAX_DPV1_SIZE);
		fbReadData(
			NETID	:= aNetId,
			PORT	:= 16#1000 + iProfibusSlaveAdr,
			IDXGRP	:= 0,
			IDXOFFS	:= 47,
			LEN		:= iMAX_DPV1_SIZE,
			DESTADDR:= pDpv1ResData,
			READ	:= FALSE,
			TMOUT	:= tTmOut,
		);
		fbReadData(READ := TRUE);
		iState	:= 3; (* CHECK READ *)
	END_IF

3:	(* wait for read response with data from DPV1 read request *)
	fbReadData(READ := FALSE);

	IF NOT fbReadData.BUSY THEN
		fbReadData(READ := FALSE);
		IF NOT fbReadData.ERR THEN
			MEMCPY(ADR(stDpv1ResHeader), pDpv1ResData, SIZEOF(stDpv1ResHeader));

			(* check for read response reference *)
			IF (stDpv1ResHeader.iRequestRef = stDpv1ReqHeader.iRequestRef) AND (stDpv1ResHeader.iAxis = stDpv1ReqHeader.iAxis) THEN
				(* response to last parameter request - split response data *)
				TmOutTimer(IN := FALSE);
				iState	:= 5; (* DONE *)
			ELSIF stDpv1ResHeader.iRequestRef = 0 THEN
				(* no response *)
				IF TmOutTimer.Q THEN
					(* complete read request timed out *)
					TmOutTimer(IN := FALSE);
					bBusy	:= FALSE;
					bError	:= TRUE;
					iErrId	:= 16#745; (* timeout *)
					iState	:= 0; (* ERROR *)
				ELSE
					(* no response, go to wait state *)
					WaitTimer(IN := FALSE);
					iState	:= 2; (* WAIT and REPEAT *)
				END_IF
			ELSE
				(* wrong response *)
				bBusy	:= FALSE;
				bError	:= TRUE;
				iErrId	:= 2; (* wrong reference response *)
				iState	:= 0; (* ERROR *)
			END_IF
		ELSE
			IF ((UDINT_TO_DWORD(fbReadData.ERRID) AND DWORD#16#FFFF0000) = DWORD#16#27B50000) THEN
				(* repeat telegram *)
				WaitTimer(IN := FALSE);
				iState	:=  4; (* SEND NEW REQUEST *)
			ELSE
				(* error *)
				bBusy	:= FALSE;
				bError	:= TRUE;
				iErrId	:= fbReadData.ERRID;
				IF ((UDINT_TO_DWORD(iErrId) AND DWORD#16#FF000000) = DWORD#16#27000000) THEN
					iErrorClass := UDINT_TO_BYTE(SHR((UDINT_TO_DWORD(iErrId) AND 16#00F00000), 20));
					iErrorCode := UDINT_TO_BYTE(SHR((UDINT_TO_DWORD(iErrId) AND 16#000F0000), 16));
				END_IF
				iState	:= 0; (* ERROR *)
			END_IF
		END_IF
	END_IF

4:	(* generate new request reference after fault *)
	WaitTimer(IN := TRUE);
	IF WaitTimer.Q THEN
		iRequestRef := UINT_TO_USINT((USINT_TO_UINT(iRequestRef) + 1) MOD 128);
		IF iRequestRef = 0 THEN
			iRequestRef := 1;
		END_IF
		pDpv1ReqData^[1] := iRequestRef;
		MEMCPY(ADR(stDpv1ReqHeader), pDpv1ReqData, SIZEOF(stDpv1ReqHeader));
	
		(* clear response data *)
		MEMSET(pDpv1ResData, 0, iMAX_DPV1_SIZE);
	
		(* send request *)
		fbWriteAccessData(
			NETID	:= aNetId,
			PORT	:= 16#1000 + iProfibusSlaveAdr,
			IDXGRP	:= 0,
			IDXOFFS	:= 47,
			LEN		:= MIN(iDpv1ReqDataLen, iMAX_DPV1_SIZE),
			SRCADDR	:= pDpv1ReqData,
			WRITE	:= FALSE,
			TMOUT	:= tTmOut
		);
		fbWriteAccessData(WRITE	:= TRUE);
	
		iState := 1; (* CHECK WRITE *)
	END_IF

5:	(* evaluate response *)
	IF stDpv1ResHeader.iRequestID = stDpv1ReqHeader.iRequestID THEN
		(* DPV1 Read successful - done *)
		bBusy	:= FALSE;
		iState	:= 0; (* DONE *)
	ELSIF (SINT_TO_BYTE(stDpv1ResHeader.iRequestID) AND 16#7F) = SINT_TO_BYTE(stDpv1ReqHeader.iRequestID) THEN
		(* DPV1 Read not successful or partly not successful *)
		bErrorValues:= TRUE;
		bBusy	:= FALSE;
		bError	:= TRUE;
		iErrId	:= 3; (* DPV1 Write not successful or partly not successful *)
		iState	:= 0; (* ERROR *)
	ELSE
		(* wrong response *)
		bBusy	:= FALSE;
		bError	:= TRUE;
		iErrId	:= 4; (* wrong response ID *)
		iState	:= 0; (* ERROR *)
	END_IF
END_CASE

(* clear flag *)
bExecute_ := bExecute_ AND bExecute;
END_FUNCTION_BLOCK

(* POU FB_Dpv1WritePNET, ST *)
FUNCTION_BLOCK FB_Dpv1WritePNET
(*****************************************************************************************************************
	DESCRIPTION:	This FUNCTION block implements DPV1 Parameter Write for Profinet

	CHANGE LOG:
	BY		DATE		DESCRIPTION OF CHANGE
	ICh		2009/07/23	First Version

******************************************************************************************************************)
VAR_INPUT
	bExecute			: BOOL;

	(* drive access info *)
	aNetId				: T_AmsNetId;	(* NetID of Profinet Master EL6631 *)
	iProfinetPort		: UINT;		 	(* Port of ProfiDrive *)
	iDriveId			: USINT;		(* 0..255 possible *)
	pDpv1ReqData		: POINTER TO ARRAY [1..iMAX_DPV1_SIZE_PNET_REQ] OF BYTE;
	iDpv1ReqDataLen		: UDINT;
	pDpv1ResData		: POINTER TO ARRAY [1..iMAX_DPV1_SIZE_PNET_RES] OF BYTE;
	iDpv1ResDataLen		: UDINT;
	tTmOut				: TIME;
END_VAR
VAR_OUTPUT
	bBusy				: BOOL;
	bError				: BOOL;
	bErrorValues		: BOOL;
	iErrId				: UDINT;
	iErrorClass			: BYTE;
	iErrorCode			: BYTE;
END_VAR
VAR_IN_OUT
	iRequestRef			: USINT;		(* 1..127;    0: reserved *)
END_VAR
VAR
	fbRWData 			: ADSRDWRT;
	iState				: INT;
	bExecute_			: BOOL;
	iIGrp				: UDINT := 16#F823;
	stDpv1ReqHeader		: ST_Dpv1Header;
	stDpv1ResHeader		: ST_Dpv1Header;
	stPNETFrameHeader	: ST_PNIOConfigRecord;

	WaitTimer			: TON := (PT := T#100ms);
	TmOutTimer			: TON;
END_VAR
TmOutTimer();

CASE iState OF
0:	(* idle until rising edge on bExecute *)
	IF bExecute AND NOT bExecute_ THEN
		(* generate request reference *)
		iRequestRef := UINT_TO_USINT((USINT_TO_UINT(iRequestRef) + 1) MOD 128);
		IF iRequestRef = 0 THEN
			iRequestRef := 1;
		END_IF
		pDpv1ReqData^[1] := 1; pDpv1ReqData^[2] := 0; (* write request *)
		pDpv1ReqData^[1+SIZEOF(stPNETFrameHeader)] := iRequestRef;
		MEMCPY(ADR(stPNETFrameHeader), pDpv1ReqData, SIZEOF(stPNETFrameHeader));
		MEMCPY(ADR(stDpv1ReqHeader), pDpv1ReqData+SIZEOF(stPNETFrameHeader), SIZEOF(stDpv1ReqHeader));

		(* clear response data *)
		MEMSET(pDpv1ResData, 0, iMAX_DPV1_SIZE_PNET_RES);

		(* on rising edge *)
		bExecute_ 	:= bExecute;
		bBusy		:= TRUE;
		bError		:= FALSE;
		bErrorValues:= FALSE;
		iErrId		:= 0;
		iErrorClass	:= 0;
		iErrorCode	:= 0;

		(* complete read request timeout 12 times the ADS timeout *)
		TmOutTimer(IN := FALSE, PT := MAX(tTmOut * 12, T#30s));
		TmOutTimer(IN := TRUE);

		(* send request *)
		fbRWData(
			NETID	:= aNetId,
			PORT	:= iProfinetPort,
			IDXGRP	:= iIGrp,
			IDXOFFS	:= 0,
			WRITELEN:= MIN(iDpv1ReqDataLen, iMAX_DPV1_SIZE_PNET_REQ),
			SRCADDR	:= pDpv1ReqData,
			READLEN	:= MIN(iDpv1ResDataLen, iMAX_DPV1_SIZE_PNET_RES),
			DESTADDR:= pDpv1ResData,
			WRTRD	:= FALSE,
			TMOUT	:= tTmOut
		);
		fbRWData(WRTRD	:= TRUE);

		iState := 1;
	END_IF

1:	(* write access data for DPV1 read request *)
	fbRWData(WRTRD	:= FALSE);

	IF NOT fbRWData.BUSY THEN
		fbRWData(WRTRD	:= FALSE);

		IF NOT fbRWData.ERR THEN
			(* read request parameter successfully sent, check for response *)
			WaitTimer(IN := FALSE);
			iState	:= 2; (* wait before polling *)
		ELSE
			bBusy	:= FALSE;
			bError	:= TRUE;
			iErrId	:= fbRWData.ERRID;
			IF ((UDINT_TO_DWORD(iErrId) AND DWORD#16#FF000000) = DWORD#16#27000000) THEN
				iErrorClass := UDINT_TO_BYTE(SHR((UDINT_TO_DWORD(iErrId) AND 16#00F00000), 20));
				iErrorCode := UDINT_TO_BYTE(SHR((UDINT_TO_DWORD(iErrId) AND 16#000F0000), 16));
			END_IF
			iState	:= 0;
		END_IF
	END_IF

2:	(* wait staate before next read response check *)
	WaitTimer(IN := TRUE);
	IF WaitTimer.Q THEN
		stPNETFrameHeader.iRW := 0; (* read response *)

		(* read request parameter successfully sent, check for read response *)
		MEMSET(pDpv1ResData, 0, iMAX_DPV1_SIZE_PNET_RES);

		fbRWData(
			NETID	:= aNetId,
			PORT	:= iProfinetPort,
			IDXGRP	:= iIGrp,
			IDXOFFS	:= 0,
			WRITELEN:= SIZEOF(stPNETFrameHeader),
			SRCADDR	:= ADR(stPNETFrameHeader),
			READLEN	:= MIN(iDpv1ResDataLen, iMAX_DPV1_SIZE_PNET_RES),
			DESTADDR:= pDpv1ResData,
			WRTRD	:= FALSE,
			TMOUT	:= tTmOut
		);
		fbRWData(WRTRD	:= TRUE);
		iState	:= 3; (* CHECK READ *)
	END_IF

3:	(* wait for read response with data from DPV1 read request *)
	fbRWData(WRTRD := FALSE);

	IF NOT fbRWData.BUSY THEN
		fbRWData(WRTRD := FALSE);
		IF NOT fbRWData.ERR THEN
			MEMCPY(ADR(stDpv1ResHeader), pDpv1ResData, SIZEOF(stDpv1ResHeader));

			(* check for read response reference *)
			IF (stDpv1ResHeader.iRequestRef = stDpv1ReqHeader.iRequestRef) AND (stDpv1ResHeader.iAxis = stDpv1ReqHeader.iAxis) THEN
				(* response to last parameter request - split response data *)
				TmOutTimer(IN := FALSE);
				iState	:= 5; (* DONE *)
			ELSIF stDpv1ResHeader.iRequestRef = 0 THEN
				(* no response *)
				IF TmOutTimer.Q THEN
					(* complete read request timed out *)
					TmOutTimer(IN := FALSE);
					bBusy	:= FALSE;
					bError	:= TRUE;
					iErrId	:= 16#745; (* timeout *)
					iState	:= 0; (* ERROR *)
				ELSE
					(* no response, go to wait state *)
					WaitTimer(IN := FALSE);
					iState	:= 2; (* WAIT and REPEAT *)
				END_IF
			ELSE
				(* wrong response *)
				bBusy	:= FALSE;
				bError	:= TRUE;
				iErrId	:= 2; (* wrong reference response *)
				iState	:= 0; (* ERROR *)
			END_IF
		ELSE
			IF ((UDINT_TO_DWORD(fbRWData.ERRID) AND DWORD#16#FFFF0000) = DWORD#16#27B50000) THEN
				(* repeat telegram *)
				WaitTimer(IN := FALSE);
				iState	:=  4; (* SEND NEW REQUEST *)
			ELSE
				(* error *)
				bBusy	:= FALSE;
				bError	:= TRUE;
				iErrId	:= fbRWData.ERRID;
				IF ((UDINT_TO_DWORD(iErrId) AND DWORD#16#FF000000) = DWORD#16#27000000) THEN
					iErrorClass := UDINT_TO_BYTE(SHR((UDINT_TO_DWORD(iErrId) AND 16#00F00000), 20));
					iErrorCode := UDINT_TO_BYTE(SHR((UDINT_TO_DWORD(iErrId) AND 16#000F0000), 16));
				END_IF
				iState	:= 0; (* ERROR *)
			END_IF
		END_IF
	END_IF

4:	(* generate new request reference after fault *)
	WaitTimer(IN := TRUE);
	IF WaitTimer.Q THEN
		iRequestRef := UINT_TO_USINT((USINT_TO_UINT(iRequestRef) + 1) MOD 128);
		IF iRequestRef = 0 THEN
			iRequestRef := 1;
		END_IF
		pDpv1ReqData^[1] := 1; pDpv1ReqData^[2] := 0; (* write request *)
		pDpv1ReqData^[1+SIZEOF(stPNETFrameHeader)] := iRequestRef;
		MEMCPY(ADR(stPNETFrameHeader), pDpv1ReqData, SIZEOF(stPNETFrameHeader));
		MEMCPY(ADR(stDpv1ReqHeader), pDpv1ReqData+SIZEOF(stPNETFrameHeader), SIZEOF(stDpv1ReqHeader));

		(* clear response data *)
		MEMSET(pDpv1ResData, 0, iMAX_DPV1_SIZE_PNET_RES);

		(* send request *)
		fbRWData(
			NETID	:= aNetId,
			PORT	:= iProfinetPort,
			IDXGRP	:= iIGrp,
			IDXOFFS	:= 0,
			WRITELEN:= MIN(iDpv1ReqDataLen, iMAX_DPV1_SIZE_PNET_REQ),
			SRCADDR	:= pDpv1ReqData,
			READLEN	:= MIN(iDpv1ResDataLen, iMAX_DPV1_SIZE_PNET_RES),
			DESTADDR:= pDpv1ResData,
			WRTRD	:= FALSE,
			TMOUT	:= tTmOut
		);
		fbRWData(WRTRD	:= TRUE);

		iState := 1; (* CHECK WRITE *)
	END_IF

5:	(* evaluate response *)
	IF stDpv1ResHeader.iRequestID = stDpv1ReqHeader.iRequestID THEN
		(* DPV1 Read successful - done *)
		bBusy	:= FALSE;
		iState	:= 0; (* DONE *)
	ELSIF (SINT_TO_BYTE(stDpv1ResHeader.iRequestID) AND 16#7F) = SINT_TO_BYTE(stDpv1ReqHeader.iRequestID) THEN
		(* DPV1 Read not successful or partly not successful *)
		bErrorValues:= TRUE;
		bBusy	:= FALSE;
		bError	:= TRUE;
		iErrId	:= 3; (* DPV1 Write not successful or partly not successful *)
		iState	:= 0; (* ERROR *)
	ELSE
		(* wrong response *)
		bBusy	:= FALSE;
		bError	:= TRUE;
		iErrId	:= 4; (* wrong response ID *)
		iState	:= 0; (* ERROR *)
	END_IF
END_CASE

(* clear flag *)
bExecute_ := bExecute_ AND bExecute;
END_FUNCTION_BLOCK

(* POU FB_GetDPRAMInfo, ST *)
FUNCTION_BLOCK FB_GetDPRAMInfo (*if the dpram must be accessed in a special manor, this function block returns error 0x701. In this case call FB_NovRamReadWriteEx to read data from the NOV-RAM and write data to the NOV-RAM.*)
VAR_INPUT
	nDevId 		: UDINT;		(* Device id of the FCxxxx or other DPRAM card ( Map the FC card as generic DPRAM/NOVRAM card im System Manager first ) *)
	bExecute		: BOOL;		(* Rising edge starts function block execution*)
	tTimeOut		: TIME := DEFAULT_ADS_TIMEOUT;	(* Max timeout for this command *)
END_VAR
VAR_OUTPUT
	bBusy 			: BOOL;
	bError			: BOOL;
	nErrid			: UDINT;
	stInfo			: ST_NovRamAddrInfo;
END_VAR
VAR
	FallingEdge		: F_TRIG;
	RisingRead		: R_TRIG;
	fbAdsReadEx	: ADSREADEX;
END_VAR
RisingRead( CLK := bExecute );
IF RisingRead.Q THEN
	bBusy := TRUE;
	bError := FALSE;
	nErrId := 0;
	MEMSET( ADR( stInfo ), 0, SIZEOF( stInfo ) );

	(* Get the nov ram address pointer and the novram byte size *)
	fbAdsReadEx( READ := FALSE );(*reset the fb*)
	fbAdsReadEx(
			NETID:= '',
			PORT:= AMSPORT_R0_IO,
			IDXGRP:= 16#5000+nDevId,
			IDXOFFS:= 16#FFFF_0200,
			LEN:= SIZEOF(stInfo),
			DESTADDR:= ADR(stInfo),
			READ:= TRUE,
			TMOUT:= tTimeout);
ELSE
		fbAdsReadEx( READ := FALSE );
END_IF

FallingEdge( CLK := fbAdsReadEx.BUSY );
IF FallingEdge.Q THEN
	bBusy := FALSE;
	IF NOT fbAdsReadEx.ERR THEN
		IF ( fbAdsReadEx.COUNT_R <> SIZEOF( stInfo ) ) THEN
			bError := TRUE;
			nErrId := 16#706;(* 1798 invalid parameter value(s)  *)
		END_IF
	ELSE
		bError := fbAdsReadEx.ERR;
		nErrId := fbAdsReadEx.ERRID;
	END_IF
END_IF
END_FUNCTION_BLOCK

(* POU FB_GetUPSStatus, ST *)
FUNCTION_BLOCK FB_GetUPSStatus
VAR_INPUT
	sNetId			: T_AmsNetId;
	nPort			: T_AmsPort := 0; (* 0 = Windows UPS service *)
	bEnable			: BOOL;
END_VAR
VAR_OUTPUT
	bValid			: BOOL;
	bError			: BOOL;
	nErrId			: UDINT;
	stStatus			:ST_UPSStatus;
END_VAR
VAR
	fbRegQueryValue : FB_RegQueryValue;
	step				: INT;
	i				: INT;
	risingEdge		: R_TRIG;
	regNames		: ARRAY[1..11] OF STRING(25):=
(*  Config REG_SZ's *)					'Model', 'Vendor',
(*  Status REG_SZ's *)					'FirmwareRev', 'SerialNumber',
(*  Status REG_DWORD's *)				'CommStatus','BatteryCapacity','BatteryStatus','TotalUPSRuntime','TcPowerFailCnt', 'TcChargeFlags','UtilityPowerStatus';
	regSZData		: STRING;
	regDWData		: DWORD;

	delay			: TON := ( PT := T#300ms);
	tTimeOut			: TIME := T#2s;
	tmpStatus		:ST_UPSStatus;
	sPort	: STRING;
	sKey	: STRING;
END_VAR
risingEdge( CLK := bEnable );
IF risingEdge.Q THEN
	delay( IN := FALSE );
	bValid := FALSE;
	bError := FALSE;
	nErrId := 0;
(*	step := 1; *)
	step := -2;
	i := 0;
	MEMSET( ADR( stStatus ), 0, SIZEOF( stStatus) );
	fbRegQueryValue( bExecute := FALSE );
ELSIF NOT bEnable THEN
	step := 0;
END_IF

CASE step OF
	-2:
		fbRegQueryValue( bExecute := FALSE );
		fbRegQueryValue(sNetId:= sNetId, sSubKey:= 'Drivers\BuiltIn\Battery', sValName:='Port', cbData:=SIZEOF(sPort) , pData:=ADR(sPort) , bExecute:= TRUE , tTimeOut:=tTimeOut );
		step := -1;

	-1:
		fbRegQueryValue( bExecute := FALSE );
		IF NOT fbRegQueryValue.bBusy THEN
			IF NOT fbRegQueryValue.bError THEN
				sKey := 'Drivers\BuiltIn\Battery';
			ELSE
				sKey := 'SYSTEM\CurrentControlSet\Services\UPS';
			END_IF

			step := 1;
		END_IF



	0:	; (* idle step *)

	1:	(* Wait some time and repeat reading...*)
		delay( IN := TRUE );
		IF delay.Q THEN
			delay( IN := FALSE );
			i := i+1;
			step := step +1;
		END_IF
	2:
		fbRegQueryValue( bExecute := FALSE );
		CASE i OF
			1..2:
				fbRegQueryValue(sNetId:= sNetId, sSubKey:= CONCAT(sKey, '\Config'), sValName:=regNames[i], cbData:=SIZEOF(regSZData) , pData:=ADR(regSZData) , bExecute:= TRUE , tTimeOut:=tTimeOut );
			3..4:
				fbRegQueryValue(sNetId:= sNetId, sSubKey:= CONCAT(sKey, '\Status'), sValName:=regNames[i], cbData:=SIZEOF(regSZData) , pData:=ADR(regSZData) , bExecute:= TRUE , tTimeOut:=tTimeOut );
			5..11:
				fbRegQueryValue(sNetId:= sNetId, sSubKey:= CONCAT(sKey, '\Status'), sValName:=regNames[i], cbData:=SIZEOF(regDWData) , pData:=ADR(regDWData) , bExecute:= TRUE , tTimeOut:=tTimeOut );
		END_CASE
		step := step +1;
	3:
		fbRegQueryValue( bExecute := FALSE );
		IF NOT fbRegQueryValue.bBusy THEN
			IF NOT fbRegQueryValue.bError THEN
				CASE i OF
					1: tmpStatus.Model := regSZData;
					2: tmpStatus.Vendor := regSZData;
					3: tmpStatus.FirmwareRev := regSZData;
					4: tmpStatus.SerialNumber := regSZData;
					5: tmpStatus.eCommStatus := DWORD_TO_INT(regDWData);
					6: tmpStatus.BatteryLifePercent := regDWData;
					7: tmpStatus.eBatteryStatus := DWORD_TO_INT(regDWData);
					8: tmpStatus.BatteryLifeTime  := regDWData;
					9: tmpStatus.nPowerFailCnt  := regDWData;
					10: tmpStatus.dwChargeFlags :=  regDWData;
					11: tmpStatus.ePowerStatus := DWORD_TO_INT(regDWData);
						stStatus := tmpStatus;
						IF ( tmpStatus.Model =  ''  ) THEN
							bValid := FALSE;
							bError := TRUE;
							nErrId := 16#8001; (*UPS configuration error (no UPS configured?)*)
						ELSIF ( tmpStatus.eCommStatus <> UpsCommOk ) THEN
							bValid := FALSE;
							bError := TRUE;
							nErrId := 16#8002; (*UPS communication error (no communication to UPS?)*)
						ELSE
							bValid := TRUE;
							bError := FALSE;
							nErrId := 0; (* no error *)
						END_IF
						i := 0;
				END_CASE
			ELSE
				bValid := FALSE;
				bError := TRUE;
				IF ( ( fbRegQueryValue.nErrId = 1 ) OR ( fbRegQueryValue.nErrId = 2 ) ) THEN
					nErrId := 16#8003; (* Unknown error reading status data (status data not preset?)*)
				ELSE
					nErrId := fbRegQueryValue.nErrId;
				END_IF
				i := i - 1;
			END_IF
			step := 1;
		END_IF
END_CASE
END_FUNCTION_BLOCK

(* POU FB_NovRamReadWrite, ST *)
FUNCTION_BLOCK FB_NovRamReadWrite (*if the dpram must be accessed in a special manor, this function block returns error 0x701. In this case use FB_NovRamReadWriteEx instead.*)
VAR_INPUT
	nDevId 	: UDINT;		(* Device id of the FCxxxx card. Map the FC card as generic DPRAM/NOVRAM card im System Manager *)
	bRead		: BOOL;		(* Rising edge starts read data block from NovRam*)
	bWrite		: BOOL;		(* Rising edge starts write data block to NovRam*)
	cbSrcLen	: UDINT;		(* Number of data bytes to write *)
	cbDestLen: UDINT;		(* Number of data bytes to read*)
	pSrcAddr	: UDINT;		(* Address of the write data buffer *)
	pDestAddr	: UDINT;		(* Address of the read data buffer *)
	tTimeOut	: TIME := DEFAULT_ADS_TIMEOUT;		(* Max timeout for this command *)
END_VAR
VAR_OUTPUT
	bBusy		: BOOL;		(* The fb is working *)
	bError		: BOOL;		(* The fb returns an error *)
	nErrId		: UDINT;		(* Error code *)
	cbRead	: UDINT;		(* Number of succesfully read data bytes *)
	cbWrite	: UDINT;		(* Number of succesfully write data bytes *)
END_VAR
VAR
	bInit			: BOOL := FALSE;
	nInitDevId		: UDINT	:= 0;
	bWantRead		: BOOL := FALSE;
	bWantWrite		: BOOL := FALSE;

	iStep			: BYTE := 0;
	RisingRead		: R_TRIG;
	RisingWrite		: R_TRIG;
	stNovRamAddrInfo: ST_NovRamAddrInfo;
	fbAdsReadEx		: ADSREADEX;
END_VAR
RisingRead( CLK := bRead );
RisingWrite( CLK := bWrite );

CASE iStep OF
0:
	(* idle step, wait for rising edge on fb input*)
	IF RisingRead.Q OR RisingWrite.Q THEN

		bBusy 	:= TRUE;
		bError 	:= FALSE;
		nErrId 	:= 0;
		cbRead 	:= 0;
		cbWrite := 0;

		bWantRead 	:=	RisingRead.Q;	(* Save flags *)
		bWantWrite 	:= 	RisingWrite.Q;

		IF	 (nDevId > 0) AND (pSrcAddr > 0) AND (cbSrcLen > 0) AND (pDestAddr > 0) AND (cbDestLen> 0) THEN

			IF 	( NOT bInit ) OR ( bInit AND ( nDevId <> nInitDevId)) THEN

				bInit := FALSE;

				nInitDevId	:= 	nDevId;	(* Save the devid *)
				MEMSET( ADR( stNovRamAddrInfo ) , SIZEOF(stNovRamAddrInfo), 0);

				(* Get the nov ram address pointer and the novram byte size *)
				fbAdsReadEx( READ := FALSE );(*reset the fb*)
				fbAdsReadEx(
						NETID:= '',
						PORT:= AMSPORT_R0_IO,
						IDXGRP:= 16#5000+nInitDevId,
						IDXOFFS:= 16#FFFF_0200,
						LEN:= SIZEOF(stNovRamAddrInfo),
						DESTADDR:= ADR(stNovRamAddrInfo),
						READ:= TRUE,
						TMOUT:= tTimeout);

				iStep := 10;	(* wait for the ads fb *)

			ELSIF bInit THEN

				IF bWantWrite THEN(* copy size bytes to novRAM *)
					cbWrite := MEMCPY(stNovRamAddrInfo.pCardAddress, pSrcAddr, MIN(cbSrcLen,stNovRamAddrInfo.iCardMemSize ) );
				END_IF
				IF bWantRead THEN(* copy size bytes from novRAM *)
					cbRead := MEMCPY(pDestAddr, stNovRamAddrInfo.pCardAddress, MIN(cbDestLen,stNovRamAddrInfo.iCardMemSize ));
				END_IF

				bBusy := FALSE;

			END_IF

		ELSE
			bBusy := FALSE;
			bError := TRUE;
			nErrId := 1798;(* invalid parameter value(s)*)
		END_IF
	END_IF

10:
	fbAdsReadEx( READ := FALSE );
	IF NOT fbAdsReadEx.BUSY THEN

		IF NOT fbAdsReadEx.ERR THEN
			bInit := TRUE;
			bError := FALSE;
			nErrId := 0;

			IF bWantWrite THEN(* copy size bytes to novRAM *)
				cbWrite := MEMCPY(stNovRamAddrInfo.pCardAddress, pSrcAddr, MIN(cbSrcLen,stNovRamAddrInfo.iCardMemSize ) );
			END_IF
			IF bWantRead THEN(* copy size bytes from novRAM *)
				cbRead := MEMCPY(pDestAddr, stNovRamAddrInfo.pCardAddress, MIN(cbDestLen,stNovRamAddrInfo.iCardMemSize ));
			END_IF
		ELSE
			bError := fbAdsReadEx.ERR;
			nErrId := fbAdsReadEx.ERRID;
		END_IF

		bBusy := FALSE;
		iStep := 0; (*go to the idle step and wait for the next call *)

	END_IF

END_CASE;
END_FUNCTION_BLOCK

(* POU FB_NovRamReadWriteEx, ST *)
FUNCTION_BLOCK FB_NovRamReadWriteEx (*if the dpram must be accessed in a special manor, this function block returns error 0x701. In this case use FB_NovRamReadWriteEx instead.*)
VAR_INPUT
	nDevId 		:	UDINT;		(* Device id of the FCxxxx card. Map the FC card as generic DPRAM/NOVRAM card im System Manager *)
	bRead		:	BOOL;		(* Rising edge starts read data block from NovRam*)
	bWrite		:	BOOL;		(* Rising edge starts write data block to NovRam*)
	cbSrcLen	:	UDINT;		(* Number of data bytes to write *)
	cbDestLen	:	UDINT;		(* Number of data bytes to read*)
	pSrcAddr	:	UDINT;		(* Address of the write data buffer *)
	pDestAddr	:	UDINT;		(* Address of the read data buffer *)
	nReadOffs	:	UDINT;		(* Offset in the DPRAM to start reading from*)
	nWriteOffs	:	UDINT;		(* Offset in the DPRAM to start writing to*)
	tTimeOut	: 	TIME;		(* Max timeout for this command *)
END_VAR
VAR_OUTPUT
	bBusy		:	BOOL;		(* The fb is working *)
	bError		:	BOOL;		(* The fb returns an error *)
	nErrId		:	UDINT;		(* Error code *)
	cbRead		: 	UDINT;		(* Number of succesfully read data bytes *)
	cbWrite		: 	UDINT;		(* Number of succesfully write data bytes *)
END_VAR
VAR
	bInit				: BOOL := FALSE;
	nInitDevId		: UDINT	:= 0;
	bWantRead		: BOOL := FALSE;
	bWantWrite		: BOOL := FALSE;
	bCopy			: BOOL := FALSE;

	i				: UDINT:=0;
	iStep			: BYTE := 0;
	RisingRead		: R_TRIG;
	RisingWrite		: R_TRIG;

	stNovRamAddrInfo	: ST_NovRamAddrInfoEx;
	fbAdsReadEx		: ADSREADEX;

	pByte			: POINTER TO BYTE;
	pCard			: POINTER TO BYTE;
END_VAR
RisingRead( CLK := bRead );
RisingWrite( CLK := bWrite );

CASE iStep OF
0:
	(* idle step, wait for rising edge on fb input*)
	IF RisingRead.Q OR RisingWrite.Q THEN

		bBusy 	:= TRUE;
		bError 	:= FALSE;
		nErrId 	:= 0;
		cbRead 	:= 0;
		cbWrite := 0;

		bWantRead 	:=	RisingRead.Q;	(* Save flags *)
		bWantWrite 	:= 	RisingWrite.Q;

		IF	(nDevId > 0) AND (  ( bWantWrite AND ( pSrcAddr>0) AND (cbSrcLen>0) ) OR ( bWantRead AND (pDestAddr > 0) AND (cbDestLen> 0) )  ) THEN
			IF 	( NOT bInit ) OR ( bInit AND ( nDevId <> nInitDevId)) THEN
				bInit := FALSE;

				nInitDevId	:= 	nDevId;	(* Save the devid *)
				MEMSET( ADR( stNovRamAddrInfo) , 10, 0);

				(* Get the nov ram address pointer and the novram byte size *)
				fbAdsReadEx( READ := FALSE );(*reset the fb*)
				fbAdsReadEx(
						NETID:= '',
						PORT:= AMSPORT_R0_IO,
						IDXGRP:= 16#5000+nInitDevId,
						IDXOFFS:= 16#FFFF_0201,
						LEN:= 10,
						DESTADDR:= ADR(stNovRamAddrInfo),
						READ:= TRUE,
						TMOUT:= tTimeout);

				iStep := 10;	(* wait for the ads fb *)

			ELSIF bInit THEN
				bCopy := TRUE;
				bBusy := FALSE;
			END_IF
		ELSE
			bBusy := FALSE;
			bError := TRUE;
			nErrId := 1798;(* invalid parameter value(s)*)
		END_IF
	END_IF

10:
	fbAdsReadEx( READ := FALSE );
	IF NOT fbAdsReadEx.BUSY THEN
		IF NOT fbAdsReadEx.ERR THEN
			bCopy := TRUE;
		ELSE
			bError := fbAdsReadEx.ERR;
			nErrId := fbAdsReadEx.ERRID;
			bBusy := FALSE;
		END_IF
		iStep := 0; (*go to the idle step and wait for the next call *)
	END_IF

END_CASE;

IF bCopy THEN
	IF  (bWantWrite AND (nWriteOffs <= stNovRamAddrInfo.iCardMemSize-1)) OR (bWantRead AND (nReadOffs <= stNovRamAddrInfo.iCardMemSize-1)) THEN
		CASE stNovRamAddrInfo.eAccessType OF
		eIOAccess_Default:
			IF bWantWrite THEN(* copy size bytes to novRAM *)
				cbWrite := MEMCPY(stNovRamAddrInfo.pCardAddress+nWriteOffs, pSrcAddr, MIN(cbSrcLen,stNovRamAddrInfo.iCardMemSize-nWriteOffs) );
			END_IF
			IF bWantRead THEN(* copy size bytes from novRAM *)
				cbRead := MEMCPY(pDestAddr, stNovRamAddrInfo.pCardAddress+nReadOffs, MIN(cbDestLen,stNovRamAddrInfo.iCardMemSize-nReadOffs));
			END_IF
		eIOAccess_Byte:
			IF bWantWrite THEN(* copy size bytes to novRAM *)
				cbWrite:=MIN(cbSrcLen,stNovRamAddrInfo.iCardMemSize-nWriteOffs);
				pByte := pSrcAddr;
				pCard := stNovRamAddrInfo.pCardAddress + nWriteOffs;
				FOR i:=1 TO cbWrite DO
					pCard^:= pByte^;
					pCard := pCard + 1;
					pByte := pByte + 1;
				END_FOR
			END_IF
			IF bWantRead THEN(* copy size bytes from novRAM *)
				cbRead:=MIN(cbDestLen,stNovRamAddrInfo.iCardMemSize-nReadOffs);
				pByte := pDestAddr;
				pCard := stNovRamAddrInfo.pCardAddress + nReadOffs;
				FOR i:=1 TO cbRead  DO
					pByte^:=pCard^;
					pCard := pCard + 1;
					pByte := pByte + 1;
				END_FOR
			END_IF
			bInit := TRUE;
			bError := FALSE;
			nErrId := 0;
		ELSE
			bInit := FALSE;
			bError := TRUE;
			nErrId := 16#701;
		END_CASE
	ELSE
		bInit := FALSE;
		bError := TRUE;
		nErrId := 16#706;
	END_IF
	bBusy := FALSE;
	bCopy:= FALSE;
END_IF
END_FUNCTION_BLOCK

(* POU FB_ReadAdsTecSysData, ST *)
FUNCTION_BLOCK FB_ReadAdsTecSysData
VAR_INPUT
	sNetId		: T_AmsNetId;
	bEnable		: BOOL;
	tCycleTime	: TIME := T#100ms;
END_VAR
VAR_OUTPUT
	bValid		: BOOL;
	bError		: BOOL;
	nErrId		: UDINT;
	stSysData	: ST_AdsTecSysData;
END_VAR
VAR
	dwTemp		: DWORD := 0;
	ptr			: POINTER TO ARRAY[0..3] OF SINT;
	delay		: TON;
	wPort		: WORD := 16#240;
	risingEdge	: R_TRIG;
	step 		: INT := 0;
	fbAdsRdWrtEx: ADSRDWRTEX;
END_VAR
risingEdge( CLK := bEnable );
IF risingEdge.Q THEN
	MEMSET( ADR( stSysData ), 0, SIZEOF( stSysData ) );
	delay( IN := FALSE, PT := tCycleTime );
	bValid := FALSE;
	bError := FALSE;
	nErrId := 0;
	step := 1;
ELSIF (NOT bEnable) THEN
	step := 0;
	bValid := FALSE;
END_IF

CASE step OF
	0:	; (* idle step *)

	1:	(* Wait some time and repeat reading...*)
		delay( IN := TRUE );
		IF delay.Q THEN
			fbAdsRdWrtEx(  WRTRD := FALSE );
			delay( IN := FALSE );
			step := step +1;
		END_IF
	2:
(*	AMSPORT_ROUTER						: UINT := 16#0001;
	ROUTERADSGRP_ACCESS_HARDWARE	: DWORD := 16#0005;
	ROUTERADSOFFS_A_HW_READIOPORT	: DWORD := 16#0001;
*)
		fbAdsRdWrtEx(  WRTRD := FALSE );
		fbAdsRdWrtEx( 	NetId := sNetId,
						Port := 1,
						IDXGRP := 16#05,
						IDXOFFS := 16#01,
						WRITELEN := SIZEOF(wPort),
						READLEN := SIZEOF(dwTemp),
						SRCADDR := ADR( wPort ),
						DESTADDR := ADR( dwTemp ),
						WRTRD := TRUE,
						TMOUT := tCycleTime
						);

		step := step +1;
	3:
		fbAdsRdWrtEx(  WRTRD := FALSE );
		IF NOT fbAdsRdWrtEx.BUSY THEN
			IF NOT fbAdsRdWrtEx.ERR THEN
				stSysData.bShiftKey := GETBIT32( dwTemp, 0 );
				stSysData.bRMouseKey := GETBIT32( dwTemp, 1 );
				stSysData.bHotkey := GETBIT32( dwTemp, 2 );
				stSysData.bTaskChaKey := GETBIT32( dwTemp, 3 );
				stSysData.bABCKey := GETBIT32( dwTemp, 4 );
				stSysData.bRsrv1 := GETBIT32( dwTemp, 5 );
				stSysData.bRsrv2 := GETBIT32( dwTemp,6 );
				stSysData.bRsrv3 := GETBIT32( dwTemp, 7 );

				stSysData.bMainFanErr := GETBIT32( dwTemp, 8 );
				stSysData.bCPUFanErr := GETBIT32( dwTemp, 9 );
				stSysData.bTempErr := GETBIT32( dwTemp, 10 );
				stSysData.bBatteryErr := GETBIT32( dwTemp, 11 );
				stSysData.bRsrv4 := GETBIT32( dwTemp, 12 );
				stSysData.bRsrv5 := GETBIT32( dwTemp, 13 );
				stSysData.bRsrv6 := GETBIT32( dwTemp, 14 );
				stSysData.bRsrv7 := GETBIT32( dwTemp, 15 );

				ptr := ADR( dwTemp );
				stSysData.nMainNTCTemp := ptr^[ 2 ];
				stSysData.nExtNTCTemp := ptr^[ 3 ];
				bValid := TRUE;
				step := 1;
			ELSE
				bValid := FALSE;
				bError := TRUE;
				nErrid := fbAdsRdWrtEx.ERRID;
				step := 0;
			END_IF
		END_IF

			;
END_CASE
END_FUNCTION_BLOCK

(* POU FB_ReadInput_analog, ST *)
(*********************************************************************************************************

NAME..............	:	FB_ReadInput_analog
DATE...............	:	11.07.2003
AUTHOR........	:	G.Sieder (Beckhoff Industrieelektronik)

DESCRIPTION:	FB for Read analog data from one Slave

HISTORY:	
11.07.2003	gs	start coding

*********************************************************************************************************)
FUNCTION_BLOCK FB_ReadInput_analog
VAR_INPUT
	iSlaveaddress		:BYTE;
	iChannel				:BYTE;
	bCycleMode			:BOOL;		(*0: Acyclic , 1:Cyclic (permanent Read/Write) *)
	bStart				:BOOL;
END_VAR
VAR_OUTPUT
	bBusy				:BOOL;
	bErr					:BOOL;
	iErrornumber			:BYTE;
	bValid				:BOOL;
	bOverflow			:BOOL;
	iReadValue			:WORD;

END_VAR
VAR_IN_OUT
	stParameterBuffer		:ST_ParameterBuffer;
END_VAR
VAR
	fbParameterinterface	:FB_ASI_Parameterinterface;
	bHiWord				:BOOL;
	iParametervalue		:DWORD;
	iParameterReadValue	:DWORD;
	iParametergroup		:WORD;
	iErrCounter			:BYTE;
	istate				:INT;
END_VAR
	CASE istate OF

		0:	IF bstart THEN
				bBusy		:=TRUE;
				bErr			:=FALSE;
				bOverflow	:=FALSE;
				bValid		:=FALSE;
				iErrornumber	:=0;
				(*check Slavenumber*)
				IF (iSlaveaddress>64) OR (iChannel>4) THEN
					bErr			:=TRUE;
					iErrornumber	:=ERROR_ASI_SLAVEADDRESS;
					istate		:=10;
				ELSE
					istate		:=1;
				END_IF
			END_IF

		(*prepare Parameternumber*)
		1:	iParametergroup	:=(iSlaveaddress*4)+(iChannel-1);
			istate	:=2;

		(*write Readrequest*)
		2:	fbParameterinterface(iParameternumber	:=iParametergroup+16#200,
							stParameterBuffer		:=stParameterBuffer,
							bParametermode		:=FALSE,
							bCycleMode			:=bCycleMode,
							bStart				:=TRUE);
			IF (NOT fbParameterinterface.bBusy) OR bCycleMode THEN
				IF fbParameterinterface.bErr THEN
					bErr			:=TRUE;
					IF fbParameterinterface.iErrornumber =1 THEN
						iErrornumber	:=ERROR_ASI_COMM_ERROR;
					ELSE
						FOR iErrCounter:=1 TO 3 DO
							IF ((SHR(fbParameterinterface.iErrornumber,iErrCounter-1)) AND 16#2000)<>0 THEN
								iErrornumber :=iErrCounter+10;
							END_IF
						END_FOR
					END_IF
					istate	:=10;
				ELSE
					IF (fbParameterinterface.iParameterReadvalue  AND 16#0200)<>0 THEN
						bOverflow	:=TRUE;
					ELSE
						bValid		:=TRUE;
					END_IF
					iParameterReadValue	:=fbParameterinterface.iParameterReadvalue;
					istate	:=3;
				END_IF
			END_IF

		(*read Parametervalue*)
		3:	iReadValue	:=DWORD_TO_WORD(iParameterReadValue);
			IF (NOT bStart) OR (NOT bCycleMode) THEN
				fbParameterinterface(bStart			:=FALSE,
								stParameterBuffer	:=stParameterBuffer);
				IF (NOT fbParameterinterface.bBusy) THEN
					istate	:=10;
				END_IF
			ELSE
				istate	:=1;
			END_IF

			(*Quit*)
		10:	bBusy	:=FALSE;
			IF (NOT bStart) THEN
				istate	:=0;
			END_IF

	ELSE
		;
	END_CASE
END_FUNCTION_BLOCK

(* POU FB_WriteOutput_analog, ST *)
(*********************************************************************************************************

NAME..............	:	FB_WriteOutput_analog
DATE...............	:	11.07.2003
AUTHOR........	:	G.Sieder (Beckhoff Industrieelektronik)

DESCRIPTION:	FB for Write analog data to one Slave

HISTORY:	
11.07.2003	gs	start coding

*********************************************************************************************************)
FUNCTION_BLOCK FB_WriteOutput_analog
VAR_INPUT
	iSlaveaddress		:BYTE;
	iChannel				:BYTE;
	iSlavevalue			:WORD;
	bCycleMode			:BOOL;		(*0: Acyclic , 1:Cyclic (permanent Read/Write) *)
	bStart				:BOOL;
END_VAR
VAR_OUTPUT
	bBusy				:BOOL;
	bErr					:BOOL;
	iErrornumber			:BYTE;

END_VAR
VAR_IN_OUT
	stParameterBuffer		:ST_ParameterBuffer;
END_VAR
VAR
	fbParameterinterface	:FB_ASI_Parameterinterface;
	bHiWord				:BOOL;
	iParametervalue		:DWORD;
	iParameterReadValue	:DWORD;
	iParametergroup		:WORD;
	iErrCounter			:BYTE;
	istate				:INT;

	iReadValue			:WORD;
END_VAR
	CASE istate OF

		0:	IF bstart THEN
				bBusy		:=TRUE;
				bErr			:=FALSE;
				iErrornumber	:=0;
				(*check Slavenumber*)
				IF (iSlaveaddress>64) OR (iChannel>4) THEN
					bErr			:=TRUE;
					iErrornumber	:=ERROR_ASI_SLAVEADDRESS;
					istate		:=10;
				ELSE
					istate		:=1;
				END_IF
			END_IF

		(*prepare Parameternumber and -value*)
		1:	iParametergroup	:=(iSlaveaddress*4)+(iChannel-1);
			iParametervalue	:=0;
			iParametervalue	:=iSlavevalue;
			iParametervalue	:=iParametervalue+16#10000;
			istate	:=2;

		(*write Parameter*)
		2:	fbParameterinterface(iParameternumber	:=iParametergroup+16#200,
							iParametervalue		:=iParametervalue,
							stParameterBuffer		:=stParameterBuffer,
							bParametermode		:=TRUE,
							bCycleMode			:=bCycleMode,
							bStart				:=TRUE);
			IF (NOT fbParameterinterface.bBusy) OR bCycleMode THEN
				IF fbParameterinterface.bErr THEN
					bErr			:=TRUE;
					IF fbParameterinterface.iErrornumber =1 THEN
						iErrornumber	:=ERROR_ASI_COMM_ERROR;
					ELSE
						FOR iErrCounter:=2 TO 4 DO
							IF ((SHR(fbParameterinterface.iErrornumber,iErrCounter-2)) AND 16#2000)<>0 THEN
								iErrornumber :=iErrCounter;
							END_IF
						END_FOR
					END_IF
					istate	:=10;
				ELSE
					iParameterReadValue	:=fbParameterinterface.iParameterReadvalue;
					istate	:=3;
				END_IF
			END_IF

		(*read Parametervalue*)
		3:	iReadValue	:=DWORD_TO_WORD(iParameterReadValue);
			IF (NOT bStart) OR (NOT bCycleMode) THEN
				fbParameterinterface(bStart			:=FALSE,
								stParameterBuffer	:=stParameterBuffer);
				IF (NOT fbParameterinterface.bBusy) THEN
					istate	:=10;
				END_IF
			ELSE
				istate	:=1;
			END_IF

			(*Quit*)
		10:	bBusy	:=FALSE;
			IF (NOT bStart) THEN
				istate	:=0;
			END_IF

	ELSE
		;
	END_CASE
END_FUNCTION_BLOCK

(* POU IOF_CAN_Layer2Command, ST *)
FUNCTION_BLOCK IOF_CAN_Layer2Command
VAR_INPUT
	NETID			: T_AmsNetId;
	DEVICEID		: UDINT;
	LEN			: UDINT;
	SRCADDR	: DWORD;
	START			: BOOL;
	TMOUT		: TIME := DEFAULT_ADS_TIMEOUT;
END_VAR
VAR_OUTPUT
	BUSY			: BOOL;
	ERR			: BOOL;
	ERRID			: UDINT;
END_VAR
VAR
	ADSWRITE1	: ADSWRITE;
	RisingEdge	: R_TRIG;
	FallingEdge	: F_TRIG;
END_VAR
RisingEdge(CLK:=START);
IF RisingEdge.Q THEN
	BUSY := TRUE;
	ERR := FALSE;
	ERRID := 0;

	IF ( DEVICEID > 0 ) AND ( MEMSET( SRCADDR, 0, LEN ) > 0 ) THEN
		ADSWRITE1(		NETID:=NETID,
						PORT:= AMSPORT_R0_IO,
						IDXGRP:= 16#00005000 +DEVICEID,
						IDXOFFS:= 16#FFFF0100,
						LEN:= LEN,
						SRCADDR:= SRCADDR,
						WRITE:=TRUE,
						TMOUT:= TMOUT );
	ELSE
		BUSY := FALSE;
		ERR := TRUE;
		ERRID := 1798; (* invalid parameter value *)
		RETURN;
	END_IF
ELSE
	ADSWRITE1( Write:=FALSE);
END_IF


FallingEdge( CLK := ADSWRITE1.BUSY );
IF FallingEdge.Q THEN
	BUSY := FALSE;
	ERR := ADSWRITE1.ERR;
	ERRID := ADSWRITE1.ERRID;
END_IF
END_FUNCTION_BLOCK

(* POU IOF_DeviceReset, ST *)
FUNCTION_BLOCK IOF_DeviceReset
VAR_INPUT
	NETID			: T_AmsNetId;
	DEVICEID		: UDINT;
	RESET		: BOOL;
	TMOUT		: TIME := DEFAULT_ADS_TIMEOUT;
END_VAR
VAR_OUTPUT
	BUSY			: BOOL;
	ERR			: BOOL;
	ERRID			: UDINT;
END_VAR
VAR
	ADSWRTCTL1: ADSWRTCTL;
	RisingEdge	: R_TRIG;
	state			: BYTE;
END_VAR
RisingEdge(CLK:=RESET);
IF RisingEdge.Q THEN
	state := 1;
END_IF
CASE state OF
	0:;(* idle state *)
	1:
		BUSY := TRUE;
		ERR := FALSE;
		ERRID := 0;
		IF ( DeviceId > 0 ) THEN
			ADSWRTCTL1( Write:=FALSE );
			ADSWRTCTL1( NETID := NETID, PORT := AMSPORT_R0_IO,
							ADSSTATE := ADSSTATE_RESET, DEVSTATE := 0,
							LEN := SIZEOF( DEVICEID ),(* if DeviceId=0xAFFE   -> reset all devices else reset only one device  *)
							SRCADDR :=ADR( DEVICEID ), Write := TRUE, TMOUT := TMOUT );
			state := 2;
		ELSE
			ERR := TRUE;
			ERRID := 16#706; (* Parameter value not correct! *)
			state := 100;
		END_IF
	2:
		ADSWRTCTL1( Write:=FALSE, BUSY=>BUSY, ERR=>ERR, ERRID=>ERRID );
		IF NOT BUSY THEN
			state := 0;
		END_IF
	100:(* error state *)
		BUSY := FALSE;
		state := 0;
END_CASE
END_FUNCTION_BLOCK

(* POU IOF_GetBoxAddrByName, ST *)
FUNCTION_BLOCK IOF_GetBoxAddrByName
VAR_INPUT
	NETID			: T_AmsNetId;
	DEVICEID		: UDINT;
	BOXNAME		: T_MaxString;
	START			: BOOL;
	TMOUT		: TIME := DEFAULT_ADS_TIMEOUT;
END_VAR
VAR_OUTPUT
	BUSY			: BOOL;
	ERR			: BOOL;
	ERRID			: UDINT;
	BOXADDR		: UINT;
END_VAR
VAR
	ADSRDWRTEX1	: ADSRDWRTEX;
	RisingEdge		: R_TRIG;
	state				: BYTE;
END_VAR
RisingEdge(CLK:=START);
IF RisingEdge.Q THEN
	state := 1;
END_IF
CASE state OF
	0:;(* idle state *)
	1:
		BUSY := TRUE;
		ERR:= FALSE;
		ERRID := 0;
		BOXADDR:=0;
		IF ( DEVICEID > 0 ) AND ( BOXNAME <> '' ) THEN
			ADSRDWRTEX1( WRTRD:=FALSE );
			ADSRDWRTEX1(	NETID:=NETID, PORT:= AMSPORT_R0_IO,
							IDXGRP:= 16#00005000 +DEVICEID, IDXOFFS:= 16#00000004,
							WRITELEN:=LEN( BOXNAME )+1, READLEN:=SIZEOF( BOXADDR ),
							SRCADDR:=ADR( BOXNAME ), DESTADDR:= ADR( BOXADDR ),
							WRTRD:=TRUE, TMOUT:= TMOUT );
			state := 2;
		ELSE
			ERR := TRUE;
			ERRID := 16#706; (* Parameter value not correct! *)
			state := 100;
		END_IF
	2:
		ADSRDWRTEX1( WRTRD:=FALSE, BUSY=>BUSY, ERR=>ERR, ERRID=>ERRID );
		IF NOT BUSY THEN
			IF NOT ERR THEN
				IF ( ADSRDWRTEX1.COUNT_R = SIZEOF( BOXADDR ) ) THEN (* check the read data length *)
					;(* OK *)
				ELSE
					ERR := TRUE;
					ERRID := 16#70B; (* 1803 invalid parameter value(s) *)
				END_IF
			END_IF
			state := 0;
		END_IF
	100:(* error state *)
		BUSY := FALSE;
		state := 0;
END_CASE
END_FUNCTION_BLOCK

(* POU IOF_GetBoxAddrByNameEx, ST *)
FUNCTION_BLOCK IOF_GetBoxAddrByNameEx
VAR_INPUT
	NETID			: T_AmsNetId;
	DEVICENAME	: T_MaxString;
	BOXNAME		: T_MaxString;
	START			: BOOL;
	TMOUT		: TIME := DEFAULT_ADS_TIMEOUT;
END_VAR
VAR_OUTPUT
	BUSY			: BOOL;
	ERR			: BOOL;
	ERRID			: UDINT;
	BOXADDR		: UINT;
END_VAR
VAR
	ADSRDWRTEX1	: ADSRDWRTEX;
	RisingEdge		: R_TRIG;
	state				: BYTE;
	StrBuff				: STRING(512);
END_VAR
RisingEdge(CLK:=START);
IF RisingEdge.Q THEN
	state := 1;
END_IF
CASE state OF
	0:;(* idle state *)
	1:
		BUSY:= TRUE;
		ERR := FALSE;
		ERRID := 0;
		BOXADDR:=0;
		IF ( DeviceName <> '' ) AND ( BoxName <> '' ) THEN
			StrBuff:=CONCAT( DeviceName, '.' );
			StrBuff:=CONCAT( StrBuff, BoxName );
			ADSRDWRTEX1( WRTRD:=FALSE );
			ADSRDWRTEX1(	NETID:=NETID, PORT:= AMSPORT_R0_IO,
							IDXGRP:= 16#00005000, IDXOFFS:= 16#00000004,
							WRITELEN:= LEN( StrBuff )+1, READLEN:=SIZEOF( BOXADDR ),
							SRCADDR:=ADR( StrBuff ), DESTADDR:= ADR( BOXADDR ),
							WRTRD:=TRUE, TMOUT:= TMOUT );
			state := 2;
		ELSE
			ERR := TRUE;
			ERRID := 16#706; (* Parameter value not correct! *)
			state := 100;
		END_IF
	2:
		ADSRDWRTEX1( WRTRD:=FALSE, BUSY=>BUSY, ERR=>ERR, ERRID=>ERRID );
		IF NOT BUSY THEN
			IF NOT ERR THEN
				IF ( ADSRDWRTEX1.COUNT_R = SIZEOF( BOXADDR ) ) THEN (* check the read data length *)
					;(* OK*)
				ELSE
					ERR := TRUE;
					ERRID := 16#70B; (* 1803 invalid parameter value(s) *)
				END_IF
			END_IF
			state := 0;
		END_IF
	100:(* error state *)
		BUSY := FALSE;
		state := 0;
END_CASE
END_FUNCTION_BLOCK

(* POU IOF_GetBoxCount, ST *)
FUNCTION_BLOCK IOF_GetBoxCount
VAR_INPUT
	NETID			: T_AmsNetId;
	DEVICEID		: UDINT;
	START			: BOOL;
	TMOUT		: TIME := DEFAULT_ADS_TIMEOUT;
END_VAR
VAR_OUTPUT
	BUSY			: BOOL;
	ERR			: BOOL;
	ERRID			: UDINT;
	BOXCOUNT	: UDINT;
END_VAR
VAR
	ADSREADEX1	: ADSREADEX;
	RisingEdge	: R_TRIG;
	state			: BYTE;
END_VAR
RisingEdge(CLK:=START);
IF RisingEdge.Q THEN
	state := 1;
END_IF
CASE state OF
	0:;(* idle state *)
	1:
		BUSY := TRUE;
		ERR:= FALSE;
		ERRID := 0;
		BOXCOUNT:=0;
		IF DEVICEID > 0 THEN
			ADSREADEX1( READ:=FALSE );
			ADSREADEX1( NETID:=NETID, PORT:= AMSPORT_R0_IO,
							IDXGRP:= 16#00005000 +DEVICEID, IDXOFFS:= 16#00000002,
							LEN:= SIZEOF( BOXCOUNT ), DESTADDR:= ADR( BOXCOUNT ),
							READ:=TRUE, TMOUT:= TMOUT );
			state := 2;
		ELSE
			ERR := TRUE;
			ERRID :=16#706;(* Parameter value not correct! *)
			state := 100;
		END_IF
	2:
		ADSREADEX1( READ:=FALSE, BUSY=>BUSY, ERR=>ERR, ERRID=>ERRID );
		IF NOT BUSY THEN
			IF NOT ERR THEN
				IF ( ADSREADEX1.COUNT_R <= SIZEOF( BOXCOUNT ) ) THEN
					;(*OK=> ChristophC: 13.08.2010-> Some 15xx builds and all TwinCAT 20xx and higher are returning only 2 bytes. Workaround: Allow 2 bytes as return length too. *)
				ELSE
					ERR := TRUE;
					ERRID := 16#70B; (* 1803 invalid parameter value(s) *)
				END_IF
			END_IF
			state := 0;
		END_IF
	100:(* error state *)
		BUSY := FALSE;
		state := 0;
END_CASE
END_FUNCTION_BLOCK

(* POU IOF_GetBoxNameByAddr, ST *)
FUNCTION_BLOCK IOF_GetBoxNameByAddr
VAR_INPUT
	NETID			: T_AmsNetId;
	DEVICEID		: UDINT;
	BOXADDR		: UINT;
	START			: BOOL;
	TMOUT		: TIME := DEFAULT_ADS_TIMEOUT;
END_VAR
VAR_OUTPUT
	BUSY			: BOOL;
	ERR			: BOOL;
	ERRID			: UDINT;
	BOXNAME		: T_MaxString;
END_VAR
VAR
	ADSRDWRTEX1	: ADSRDWRTEX;
	RisingEdge		: R_TRIG;
	state				: BYTE;
END_VAR
RisingEdge(CLK:=START);
IF RisingEdge.Q THEN
	state := 1;
END_IF
CASE state OF
	0:;(* idle state *)
	1:
		BUSY:=TRUE;
		ERR:=FALSE;
		ERRID := 0;
		MEMSET( ADR( BOXNAME ), 0, SIZEOF( BOXNAME ) );
		IF ( DEVICEID > 0 ) AND ( BOXADDR > 0 ) THEN
			ADSRDWRTEX1( WRTRD:=FALSE );
			ADSRDWRTEX1(	NETID:=NETID, PORT:= AMSPORT_R0_IO,
							IDXGRP:= 16#00005000 + DEVICEID, IDXOFFS:= 16#00000003,
							WRITELEN:= SIZEOF( BOXADDR ), READLEN:=SIZEOF( BOXNAME ) - 1, (* saves termination byte *)
							SRCADDR:=ADR( BOXADDR ), DESTADDR:= ADR( BOXNAME ),
							WRTRD:=TRUE, TMOUT:= TMOUT );
			state := 2;
		ELSE
			ERR := TRUE;
			ERRID := 16#706;(* Parameter value not correct! *)
			state := 100;
		END_IF
	2:
		ADSRDWRTEX1( WRTRD:=FALSE, BUSY=>BUSY, ERR=>ERR, ERRID=>ERRID );
		IF NOT BUSY THEN
			state := 0;
		END_IF
	100:(* error state *)
		BUSY := FALSE;
		state := 0;
END_CASE
END_FUNCTION_BLOCK

